	FB_AlarmCodeManager(	
		bAlarm1			:= MesDataExd.MesData.ProtectRelay_FeederMVCB[1].OUT_CmdOpen , 	// ProtectRelay_FeederMVCB Midi : Cmd Open
		bAlarm2			:= MesDataExd.MesData.ProtectRelay_FeederMVCB[1].OUT_CmdClose,     // ProtectRelay_FeederMVCB Midi  : Cmd Close
		bAlarm3			:= MesDataExd.MesData.ProtectRelay_FeederMVCB[2].OUT_CmdOpen  ,    // ProtectRelay_FeederMVCB Plat  : Cmd Open
		bAlarm4			:= MesDataExd.MesData.ProtectRelay_FeederMVCB[2].OUT_CmdClose ,	// ProtectRelay_FeederMVCB Plat  : Cmd Close
		bAlarm5			:= MesDataExd.MesData.TapChanger.OUT_CmdRampUp,					// 225 kV Regleur : Cmd Ramp Up
		bAlarm6			:= MesDataExd.MesData.TapChanger.OUT_CmdRampDown ,                 // 225 kV Regleur :	Cmd Ramp Down
		bAlarm7			:= MesDataExd.MesData.MesAuxHtOpenSectLine225kV	 ,				// Aux Ht : Sect Line 225 kV Open
		bAlarm8			:= MesDataExd.MesData.MesAuxHtCloseSectLine225kV	,               // Aux Ht : Sect Line 225 kV Close
		bAlarm9			:= MesDataExd.MesData.MesAuxHtTeleCondamnSl225kV	 ,				// Aux Ht : Tele Condamn Sl 225 kV 
		bAlarm10		:= MesDataExd.MesData.MesAuxHtDeTeleCondamnSl225kV,       		// Aux Ht : DeTele Condamn Sl 225 kV
		bAlarm11		:= MesDataExd.MesData.MesAuxHtTelecommandeRelestActif ,			// Aux Ht : Telecommande Relest Actif
		bAlarm12		:= MesDataExd.MesData.MesAuxHtTelecommandeRelestPassif,           // Aux Ht : Telecommande Relest Passif
		bAlarm13		:= FALSE,
		bAlarm14		:= FALSE,
		bAlarm15		:= FALSE,
		wAlarmCode		=>MesDataExd.MesData.MesEventCode2);	
		
		
	FB_AlarmCodeManager(
		bAlarm1			:= MesDataExd.MesData.MesAuxHtOpenSectMalt,				// Aux Ht Sect Malt : Open
		bAlarm2			:= MesDataExd.MesData.MesAuxHtCloseSectMalt,				// Aux Ht Sect Malt : Close
		bAlarm3			:= MesDataExd.MesData.MesAuxBtSyntOpenDistrib48VccJdb,		// Aux Bt Synt : Open Distrib 48 Vcc Jdb
		bAlarm4			:= MesDataExd.MesData.MesAuxBtSyntOpenDistrib48VccLocker,	// Aux Bt Synt : Open Distrib 48 Vcc Locker
		bAlarm5			:= MesDataExd.MesData.MesAuxBt400VPermutAutoStopMode	,	// Aux Bt 400 V Permut Auto Stop Mode				
		bAlarm6			:= MesDataExd.MesData.MesAuxBt400VPermutAutoNormalMode	 ,	// Aux Bt 400 V Permut Auto Normal Mode
		bAlarm7			:= MesDataExd.MesData.MesAuxBt400VPermutAutoSecoursMode,	// Aux Bt 400 V Permut Auto Secours Mode
		bAlarm8			:= MesDataExd.MesData.MesAuxBt400VPermutModeAuto	,		// Aux Bt 400 V Permut Mode Auto
		bAlarm9			:= MesDataExd.MesData.UPS_CE.MesOpened_CBRectifier	,		// UPC CE : Opened CB Rectifier
		bAlarm10		:= MesDataExd.MesData.UPS_CE.MesOpened_CBBatt		    ,	// UPC CE : Opened CB Batt
		bAlarm11		:= MesDataExd.MesData.UPS_CE.MesOpened_CBAntenna		 ,	// UPC CE : Opened CB Antenna
		bAlarm12		:= MesDataExd.MesData.UPS_TCM.MesOpened_CBRectifier	,	// UPC TCM : Opened CB Rectifier
		bAlarm13		:= MesDataExd.MesData.UPS_TCM.MesOpened_CBBatt	   	 ,		// UPC TCM : Opened CB Batt
		bAlarm14		:= MesDataExd.MesData.UPS_TCM.MesOpened_CBAntenna	  ,		// UPC TCM : Opened CB Antenna 
		bAlarm15		:= FALSE,//  
		wAlarmCode		=>MesDataExd.MesData.MesEventCode3);
END_METHOD

METHOD M_CP
//////////////////
//  Emulator
/////////////////

VAR 
	// Method local variables (reinitialized at each cycle) 
	

END_VAR
Trig_Cmd_Read(CLK:=IN_CmdToggleRead);


IF Trig_Cmd_Read.Q THEN
	IN_CmdToggleRead := FALSE;
MesDataExd.MesData.MesCP_Read := NOT MesDataExd.MesData.MesCP_Read;
END_IF
END_METHOD

METHOD M_Execute
//////////////////
//  Method Calls 
/////////////////
VAR 
	// Method local variables (reinitialized at each cycle) 
	// EMULATOR

	
END_VAR
// READING AND WRITING CLOCK //
	TP1(IN:=NOT TP1.Q , PT:= ParamClockReadTime);
	ClockRead 		:= TP1.Q;
	
// METHODS CALLS //

	M_Read() ; 
	M_CP();
	
// EVALUATE  /////////////
	

	
	////////////////////
	M_AlarmManagement();
END_METHOD

METHOD M_Read : BOOL
VAR_INPUT
END_VAR
VAR
	MW					: FB_MergeWordsToDint;
END_VAR
// CP-Read / Write 

MesDataExd.MesData.MesCP_Read := MesCP_Read ; 
MesDataExd.MesData.MesCP_Write := MesCP_Write ;  

IF MesCP_Read  THEN	

	// Analogic Inputs Modbus Requests
	
	FB_ModbusReadAI[1](pDestAddr := ADR(AI_List_1),
					sIPAddr := ParamIPAdr,
					tTimeout := ParamTimeout,
					nTcpPort := 502,
					nQuantity := 123,
					nMBAddr := 593,
					cbLength := SIZEOF(AI_List_1),
					nUnitID := 1,
					ClockRead := ClockRead,
					Reset := IN_CmdReset_L);
					
	FB_ModbusReadAI[2](pDestAddr := ADR(AI_List_2),
					sIPAddr := ParamIPAdr,
					tTimeout := ParamTimeout,
					nTcpPort := 502,
					nQuantity := 97,
					nMBAddr := 721,
					cbLength := SIZEOF(AI_List_2),
					nUnitID := 1,
					ClockRead := ClockRead,
					Reset := IN_CmdReset_L);
					
	// Digital Inputs Modbus Requests 
	
	FB_ModbusReadDI[1](pDestAddr := ADR(DI_List_1),
					sIPAddr := ParamIPAdr,
					tTimeout := ParamTimeout,
					nTcpPort := 502,
					nQuantity := 1683,
					nMBAddr := 480,
					cbLength := SIZEOF(DI_List_1),
					nUnitID := 1,
					ClockRead := ClockRead,
					Reset := IN_CmdReset_L);
					
	FB_ModbusReadDI[2](pDestAddr := ADR(DI_List_2),
					sIPAddr := ParamIPAdr,
					tTimeout := ParamTimeout,
					nTcpPort := 502,
					nQuantity := 1249,
					nMBAddr := 5072,
					cbLength := SIZEOF(DI_List_2),
					nUnitID := 1,
					ClockRead := ClockRead,
					Reset := IN_CmdReset_L);
	
					
					
	//  MesDataExd.MesData.Filling Digital Data				
	
MesDataExd.MesData.ProtectRelay_MainHVCB.MesAlarm_Phase1			:= DI_List_1[1]   ;
MesDataExd.MesData.ProtectRelay_MainHVCB.MesAlarm_Phase2		    := DI_List_1[2]   ;
MesDataExd.MesData.ProtectRelay_MainHVCB.MesAlarm_Phase3			:= DI_List_1[3]   ;
MesDataExd.MesData.ProtectRelay_MainHVCB.MesAlarm_PhaseRpt			:= DI_List_1[33]  ;
MesDataExd.MesData.ProtectRelay_MainHVCB.MesAlarm_Ground			:= DI_List_1[35]  ;
MesDataExd.MesData.ProtectRelay_MainHVCB.MesAlarm_GroundRpt		:= DI_List_1[36]  ;
MesDataExd.MesData.ProtectRelay_MainHVCB.MesAlarm_MaxUInverse		:= DI_List_1[37]  ;
MesDataExd.MesData.ProtectRelay_MainHVCB.MesAlarm_MaxP				:= DI_List_1[38]  ;
MesDataExd.MesData.ProtectRelay_MainHVCB.MesAlarm_CB				:= DI_List_1[39]  ;	
MesDataExd.MesData.ProtectRelay_MainHVCB.MesAlarm_Watchdog			:= DI_List_1[148] ;
	
				
	MesDataExd.MesData.ProtectRelay_Transfo225kV.MesAlarm_DiscordSectLigneHTB		   := DI_List_1[164]    ;
	MesDataExd.MesData.ProtectRelay_Transfo225kV.MesAlarm_DiscordSectMaltHTB         := DI_List_1[165]    ;
	MesDataExd.MesData.ProtectRelay_Transfo225kV.MesAlarm_DiscordSectDisjHTB         := DI_List_1[166]    ;
	MesDataExd.MesData.ProtectRelay_Transfo225kV.MesAlarm_TeleCondamne               := DI_List_1[167]    ;
	MesDataExd.MesData.ProtectRelay_Transfo225kV.MesAlarm_DeTeleCondamne             := DI_List_1[168]    ;
	MesDataExd.MesData.ProtectRelay_Transfo225kV.MesAlarm_DiscordTeleCondamne	       := DI_List_1[169]    ;
	MesDataExd.MesData.ProtectRelay_Transfo225kV.MesDataExd.MesData.MesAlarmImax                := DI_List_1[171]    ;
	MesDataExd.MesData.ProtectRelay_Transfo225kV.MesAlarm_IoMaxCoteProd              := DI_List_1[172]    ;
	MesDataExd.MesData.ProtectRelay_Transfo225kV.MesDataExd.MesData.MesAlarmUmin                := DI_List_1[173]    ;
	MesDataExd.MesData.ProtectRelay_Transfo225kV.MesDataExd.MesData.MesAlarmUmin_Long           := DI_List_1[174]    ;
	MesDataExd.MesData.ProtectRelay_Transfo225kV.MesAlarmUMax                        := DI_List_1[175]    ;
	MesDataExd.MesData.ProtectRelay_Transfo225kV.MesAlarmUMax_Long                   := DI_List_1[176]    ;
	MesDataExd.MesData.ProtectRelay_Transfo225kV.MesAlarm_PhaseRpt           	 	   := DI_List_1[177]    ;
	MesDataExd.MesData.ProtectRelay_Transfo225kV.MesWarning_ImgTherm                 := DI_List_1[178]    ;
	MesDataExd.MesData.ProtectRelay_Transfo225kV.MesAlarm_ImgTherm                   := DI_List_1[179]    ;
	MesDataExd.MesData.ProtectRelay_Transfo225kV.MesAlarm_DifferTransfo              := DI_List_1[180]    ;
	MesDataExd.MesData.ProtectRelay_Transfo225kV.MesAlarm_FreqMax                    := DI_List_1[181]    ;
	MesDataExd.MesData.ProtectRelay_Transfo225kV.MesAlarm_FreqMin                    := DI_List_1[183]    ;
	
	
	MesDataExd.MesData.MainHVCB.MesDataExd.MesData.MesClosed            				:= DI_List_1[193]    ;
	MesDataExd.MesData.MainHVCB.MesAlarm_SF6              				:= DI_List_1[197]    ;
	MesDataExd.MesData.MainHVCB.MesAlarm_Disarmed             	 		:= DI_List_1[198]    ;
	MesDataExd.MesData.MainHVCB.MesComutLocal         			   		:= DI_List_1[199]    ;
	MesDataExd.MesData.MainHVCB.MesAlarm_ArmingMotor           			:= DI_List_1[200]    ;
	MesDataExd.MesData.MainHVCB.MesAlarm_230V           					:= DI_List_1[201]    ;
	MesDataExd.MesData.MainHVCB.MesAlarmPwr          			 			:= DI_List_1[202]    ;
	
	MesDataExd.MesData.Transfo_225kV.MesWarningGas               			:= DI_List_1[220]    ;
	MesDataExd.MesData.Transfo_225kV.MesDataExd.MesData.MesAlarmGas           	 	:= DI_List_1[221]    ;
	MesDataExd.MesData.Transfo_225kV.MesDataExd.MesData.MesWarningTemp               := DI_List_1[222]    ;
	MesDataExd.MesData.Transfo_225kV.MesDataExd.MesData.MesAlarmGas             		:= DI_List_1[223]    ;
	MesDataExd.MesData.Transfo_225kV.MesWarning_TempLevel1           		:= DI_List_1[224]    ;
	MesDataExd.MesData.Transfo_225kV.MesWarning_TempLevel2          		:= DI_List_1[225]    ;
	MesDataExd.MesData.Transfo_225kV.MesTrigger_Deletion            		:= DI_List_1[228]    ;
	MesDataExd.MesData.Transfo_225kV.MesAlarm_OilLevel              		:= DI_List_1[229]    ;
	MesDataExd.MesData.Transfo_225kV.MesTransfoRefrigLocal                := DI_List_1[230]    ;
	MesDataExd.MesData.Transfo_225kV.MesTrigger_NonReturnValve       		:= DI_List_1[231]    ;
	MesDataExd.MesData.Transfo_225kV.MesTrigger_ProtectRelay      		:= DI_List_1[232]    ;
	MesDataExd.MesData.Transfo_225kV.MesAlarm_TapChanger            		:= DI_List_1[233]    ;
	
	MesDataExd.MesData.Mes20kVCourNeutCuveDefaultMasseCuve1		:= DI_List_1[305]	;
	MesDataExd.MesData.Mes20kVCourNeutCuveMaxIexp2				:= DI_List_1[306]   ;
	MesDataExd.MesData.Mes20kVCourNeutCuveDefaultMasseCuve2  		:= DI_List_1[307]   ;
	MesDataExd.MesData.Mes20kVCourNeutCuveMaxIexp4				:= DI_List_1[308]   ;
	MesDataExd.MesData.Mes20kVCourNeutCuveDefaultGround	    	:= DI_List_1[309]   ;
	MesDataExd.MesData.Mes20kVCourNeutCuveMaxI0exp4		    	:= DI_List_1[310]   ;
	MesDataExd.MesData.Mes20kVCourNeutCuveTempAlarm		    	:= DI_List_1[439]   ;
	MesDataExd.MesData.Mes20kVCourNeutCuveTempTrigger				:= DI_List_1[440]   ;
	MesDataExd.MesData.Mes20kVCourNeutCuveGazDischarge			:= DI_List_1[441]   ;
	MesDataExd.MesData.Mes20kVCourNeutCuvePressure           		:= DI_List_1[442]   ;
	
	MesDataExd.MesData.ProtectRelay_MainMVCB.MesAlarm_Phase1 			:= DI_List_1[457]	;
	MesDataExd.MesData.ProtectRelay_MainMVCB.MesAlarm_Phase2			:= DI_List_1[459]   ; // Phase 3  ? 
	MesDataExd.MesData.ProtectRelay_MainMVCB.MesAlarm_CB 				:= DI_List_1[495]   ;
	MesDataExd.MesData.ProtectRelay_MainMVCB.MesDataExd.MesData.MesTripped 		:= DI_List_1[586]   ; // Mes20kVGeneralHVCellProtectCircuitBreaker
	 /  MesDataExd.MesData.Mes20kVGeneralHVCellDefaultFrom225kV			:= DI_List_1[592]   ;
	
	MesDataExd.MesData.ProtectRelay_FeederMVCB[1].MesDataExd.MesData.MesAlarmImax 							:=	DI_List_1[609]	;
	MesDataExd.MesData.ProtectRelay_FeederMVCB[1].MesAlarm_MaxP									:=	DI_List_1[611]  ;
	MesDataExd.MesData.ProtectRelay_FeederMVCB[1].MesAlarm_Ground									:=	DI_List_1[613]  ;
	//  MesDataExd.MesData.AX_ProtectRelay_FeederMVCB[1].Mes20kVMidiSepamDefaultCablesOvercharge	:=	DI_List_1[641]  ;
	//  MesDataExd.MesData.AX_ProtectRelay_FeederMVCB[1].Mes20kVMidiHVCellDefaultFrom225kV			:=	DI_List_1[647]  ;
	MesDataExd.MesData.ProtectRelay_FeederMVCB[1].MesDataExd.MesData.MesTripped								:=	DI_List_1[738]  ;
	                                                                                	
	MesDataExd.MesData.ProtectRelay_FeederMVCB[2].MesDataExd.MesData.MesAlarmImax							:=	 DI_List_1[761] ;
	MesDataExd.MesData.ProtectRelay_FeederMVCB[2].MesAlarm_MaxP									:=   DI_List_1[763] ;
	MesDataExd.MesData.ProtectRelay_FeederMVCB[2].MesAlarm_Ground									:=   DI_List_1[765] ;  
	//  MesDataExd.MesData.AX_ProtectRelay_FeederMVCB[2].Mes20kVMidiSepamDefaultCablesOvercharge	:=   DI_List_1[793] ;
	//  MesDataExd.MesData.AX_ProtectRelay_FeederMVCB[2].Mes20kVMidiHVCellDefaultFrom225kV			:=   DI_List_1[799] ;
	MesDataExd.MesData.ProtectRelay_FeederMVCB[2].MesDataExd.MesData.MesTripped								:=   DI_List_1[890] ;
	
	MesDataExd.MesData.TapChanger.MesAlarm  := DI_List_1[1065] ;
	
	MesDataExd.MesData.MesAuxHTSect225kV							:=	DI_List_1[1217]	 ;
	MesDataExd.MesData.MesAuxHtSmaltHTBOpen						:=	DI_List_1[1219]	 ;
	MesDataExd.MesData.MesAuxHtFusionFuseMeasures225kV			:=	DI_List_1[1225]	 ;
	MesDataExd.MesData.MesAuxHtFusionFuseProtect225kV				:=	DI_List_1[1226]	 ;
	MesDataExd.MesData.MesAuxHtFusionFuseCountRte225kV			:=	DI_List_1[1227]	 ;
	MesDataExd.MesData.MesAuxHtShortCircuitCurrentProtectCcp2		:=	DI_List_1[1228]	 ;
	MesDataExd.MesData.MesAuxHtDisjCount20kVOpen					:=	DI_List_1[1230]	 ;
	MesDataExd.MesData.MesAuxHtDisjRefVoltage20kVOpen				:=	DI_List_1[1231]	 ;
	MesDataExd.MesData.MesAuxHtShortCircuitCurrentProtectCcp3		:=	DI_List_1[1232]	 ;
	MesDataExd.MesData.MesAuxBtTriggerGeneralDisj					:=	DI_List_1[1372]	 ;
	MesDataExd.MesData.MesAuxBt400VManqueAC						:=	DI_List_1[1373]	 ;
	MesDataExd.MesData.MesAuxBt400VDecltAntenneScada				:=	DI_List_1[1374]  ;
	MesDataExd.MesData.MesAuxBt400VDecltAntennePrio				:=	DI_List_1[1375]	 ;
	MesDataExd.MesData.MesAuxBt400VPermutAutoStopMode				:=	DI_List_1[1377]	 ;
	MesDataExd.MesData.MesAuxBt400VPermutAutoNormalMode			:=	DI_List_1[1378]	 ;
	MesDataExd.MesData.MesAuxBt400VPermutAutoSecoursMode			:=	DI_List_1[1379]	 ;
	MesDataExd.MesData.MesAuxBt400VPermutModeAuto					:=	DI_List_1[1380]	 ;
	MesDataExd.MesData.MesAuxBt400VVoltageLossNormalAlim			:=	DI_List_1[1381]	 ;
	MesDataExd.MesData.MesAuxBt400VVoltageLossSecoursAlim			:=	DI_List_1[1382]	 ;
	MesDataExd.MesData.MesAuxBt400VDefaultPermut					:=	DI_List_1[1383]	 ;
	
	
	
	MesDataExd.MesData.UPS_CE.MesAlarm_Batt 						:=	DI_List_1[1384]	 ;
	MesDataExd.MesData.UPS_CE.MesDataExd.MesData.MesAlarmState 				:=	DI_List_1[1385]	 ;
	MesDataExd.MesData.UPS_CE.MesAlarm_IsolBatt					:=	DI_List_1[1386]	 ;
	MesDataExd.MesData.UPS_CE.MesOpened_CBRectifier				:=	DI_List_1[1387]	 ;
	MesDataExd.MesData.UPS_CE.MesOpened_CBBatt					:=	DI_List_1[1388]	 ;
	MesDataExd.MesData.UPS_CE.MesOpened_CBAntenna					:=	DI_List_1[1389]	 ;
	MesDataExd.MesData.UPS_TCM.MesAlarm_Batt						:=	DI_List_1[1390]	 ;
	MesDataExd.MesData.UPS_TCM.MesDataExd.MesData.MesAlarmState				:=	DI_List_1[1391]	 ;
	MesDataExd.MesData.UPS_TCM.MesOpened_CBRectifier				:=	DI_List_1[1392]	 ;
	MesDataExd.MesData.UPS_TCM.MesOpened_CBBatt	   				:=	DI_List_1[1393]	 ;
	MesDataExd.MesData.UPS_TCM.MesOpened_CBAntenna				:=	DI_List_1[1394]	 ;
	 
	MesDataExd.MesData.MesAuxBtDefaultInverter					:=	DI_List_1[1395]	 ;
	MesDataExd.MesData.MesAuxBtSyntDefaultDistrib48VccJdb			:=	DI_List_1[1397]	 ;
	MesDataExd.MesData.MesAuxBtSyntOpenDistrib48VccJdb			:=	DI_List_1[1398]	 ;
	MesDataExd.MesData.MesAuxBtSyntDefaultDistrib48VccLocker		:=	DI_List_1[1403]	 ;
	MesDataExd.MesData.MesAuxBtSyntOpenDistrib48VccLocker			:=	DI_List_1[1404]	 ;
	 
	MesDataExd.MesData.Transfo_Aux.MesDataExd.MesData.MesAlarmTemp			:=	DI_List_1[1522]	 ;
	MesDataExd.MesData.Transfo_Aux.MesDataExd.MesData.MesAlarmGas			:=	DI_List_1[1523]	 ;
	MesDataExd.MesData.Transfo_Aux.MesDataExd.MesData.MesAlarmOilLevel		:=	DI_List_1[1524]	 ;
	 
	MesDataExd.MesData.MesAuxTransfoMeltingFusesContact			:=	DI_List_1[1525]	 ;                             
	MesDataExd.MesData.MesAuxTransfoSwitchGear	            	:=	DI_List_1[1526]  ;
	
	MesDataExd.MesData.DS.MesAlarmState          	  	:=	DI_List_1[1673] ;
	MesDataExd.MesData.FSS.MesAlarmFire				:=	DI_List_1[1674]	;
	MesDataExd.MesData.MesLocalRemoteOperation  	:=	DI_List_1[1682]	;
	MesDataExd.MesData.ES.MesAlarmState         		:=	DI_List_1[1683]	;
	 
	
						
	 /  MesDataExd.MesData.ProtectRelay_MainHVCB.MesDataExd.MesData.MesWatchdog 	  := DI_List_2[1]	; 
	MesDataExd.MesData.ProtectRelay_MainHVCB.MesDataExd.MesData.MesAlarmTCS    := DI_List_2[12]	;
	
	MesDataExd.MesData.ProtectRelay_Transfo225kV.MesDataExd.MesData.MesAlarmTCS 	 := DI_List_2[39] ;
	 // Mes225kVTransfoDefaultInternDisjCde := DI_List_2[46] ;
	
	MesDataExd.MesData.ProtectRelay_MainMVCB.MesDataExd.MesData.MesWatchdog 	 :=   DI_List_2[97]	; 
	MesDataExd.MesData.ProtectRelay_MainMVCB.MesDataExd.MesData.MesAlarmTCS   := 	DI_List_2[108]	;
	
	MesDataExd.MesData.ProtectRelay_FeederMVCB[1].MesDataExd.MesData.MesWatchdog   :=   DI_List_2[129] ;
	MesDataExd.MesData.ProtectRelay_FeederMVCB[1].MesDataExd.MesData.MesAlarmTCS   := 	 DI_List_2[140] ;
	
	MesDataExd.MesData.ProtectRelay_FeederMVCB[2].MesDataExd.MesData.MesWatchdog	  :=   DI_List_2[161]  ; 
	MesDataExd.MesData.ProtectRelay_FeederMVCB[2].MesDataExd.MesData.MesAlarmTCS   := 	 DI_List_2[172]  ;
	
	MesDataExd.MesData.TapChanger.MesAlarm_Discordance				  :=  DI_List_2[225]	;
	MesDataExd.MesData.TapChanger.MesAlarm_NoOutletDetected			  :=  DI_List_2[226]	;          
	MesDataExd.MesData.TapChanger.MesModeAuto							  :=  DI_List_2[227]	;
	MesDataExd.MesData.TapChanger.MesModeManual						  :=  DI_List_2[228]	;
	MesDataExd.MesData.TapChanger.MesState_ManoeuverAuthorized 		  :=  DI_List_2[230]	;
	
	MesDataExd.MesData.ProtectRelay_MainHVCB.OUT_CmdOpen  			  :=  DI_List_2[990] ;
	MesDataExd.MesData.ProtectRelay_MainHVCB.OUT_CmdClose     		  :=  DI_List_2[991] ;
	
	//  MesDataExd.MesData.Mes225kVTransfoDeclenchOpen	 := DI_List_2[1019] ;
	//  MesDataExd.MesData.Mes225kVTransfoEnclenchClose    := DI_List_2[1020] ;
	
	MesDataExd.MesData.ProtectRelay_MainMVCB.OUT_CmdOpen 	 :=  DI_List_2[1077] ;
	MesDataExd.MesData.ProtectRelay_MainMVCB.OUT_CmdClose  :=  DI_List_2[1078] ;
	
	MesDataExd.MesData.ProtectRelay_FeederMVCB[1].OUT_CmdOpen 	:=	DI_List_2[1106]  ; // MIDI 
	MesDataExd.MesData.ProtectRelay_FeederMVCB[1].OUT_CmdClose :=  DI_List_2[1107]  ;
	
	MesDataExd.MesData.ProtectRelay_FeederMVCB[2].OUT_CmdOpen   :=  DI_List_2[1135]	;	// PLAT 
	MesDataExd.MesData.ProtectRelay_FeederMVCB[2].OUT_CmdClose  :=  DI_List_2[1136]  ;
	
	MesDataExd.MesData.TapChanger.OUT_CmdRampUp	:=  DI_List_2[1193] ;
	MesDataExd.MesData.TapChanger.OUT_CmdRampDown :=	DI_List_2[1194] ;           
	MesDataExd.MesData.TapChanger.MesModeManual	:=  DI_List_2[1195]	;
	MesDataExd.MesData.TapChanger.MesModeAuto    :=  DI_List_2[1196] ;
	
	MesDataExd.MesData.MesAuxHtOpenSectLine225kV		  :=  DI_List_1[1242]  	;
	MesDataExd.MesData.MesAuxHtCloseSectLine225kV		  :=  DI_List_1[1243] 	;
	MesDataExd.MesData.MesAuxHtOpenSectMalt			  :=  DI_List_1[1244]   ;  
	MesDataExd.MesData.MesAuxHtCloseSectMalt			  :=  DI_List_1[1245]   ; 	
	MesDataExd.MesData.MesAuxHtTeleCondamnSl225kV		  :=  DI_List_1[1246] 	;
	MesDataExd.MesData.MesAuxHtDeTeleCondamnSl225kV	  :=  DI_List_1[1247]   ;                          
	MesDataExd.MesData.MesAuxHtTelecommandeRelestActif  :=  DI_List_1[1248]   ;
	MesDataExd.MesData.MesAuxHtTelecommandeRelestPassif :=  DI_List_1[1249]   ;
	
	//  MesDataExd.MesData.Filling Analogic Data			           
					                                
	MW(WORD_STRONG :=  AI_List_1[1  ],	WORD_WEAK := AI_List_1[1  ], SIZE := 1, FIX := 0, SIGNED := 0, VAR_OUT	:= MesDataExd.MesData.ProtectRelay_MainHVCB.MesDataExd.MesData.MesI1);
	MW(WORD_STRONG :=  AI_List_1[2  ],	WORD_WEAK := AI_List_1[2  ], SIZE := 1, FIX := 0, SIGNED := 0, VAR_OUT	:= MesDataExd.MesData.ProtectRelay_MainHVCB.MesDataExd.MesData.MesI2);
	MW(WORD_STRONG :=  AI_List_1[3  ],	WORD_WEAK := AI_List_1[3  ], SIZE := 1, FIX := 0, SIGNED := 0, VAR_OUT	:= MesDataExd.MesData.ProtectRelay_MainHVCB.MesDataExd.MesData.MesI3);
	MW(WORD_STRONG :=  AI_List_1[12 ],	WORD_WEAK := AI_List_1[12 ], SIZE := 1, FIX := 3, SIGNED := 0, VAR_OUT	:= MesDataExd.MesData.ProtectRelay_MainHVCB.MesDataExd.MesData.MesU12);
	MW(WORD_STRONG :=  AI_List_1[13 ],	WORD_WEAK := AI_List_1[13 ], SIZE := 1, FIX := 3, SIGNED := 0, VAR_OUT	:= MesDataExd.MesData.ProtectRelay_MainHVCB.MesDataExd.MesData.MesU23);
	MW(WORD_STRONG :=  AI_List_1[14 ],	WORD_WEAK := AI_List_1[14 ], SIZE := 1, FIX := 3, SIGNED := 0, VAR_OUT	:= MesDataExd.MesData.ProtectRelay_MainHVCB.MesDataExd.MesData.MesU31);
	MW(WORD_STRONG :=  AI_List_1[18 ],	WORD_WEAK := AI_List_1[18 ], SIZE := 1, FIX := 0, SIGNED := 0, VAR_OUT	:= MesDataExd.MesData.ProtectRelay_MainHVCB.MesU0);
	MW(WORD_STRONG :=  AI_List_1[21 ],	WORD_WEAK := AI_List_1[21 ], SIZE := 1, FIX := 0, SIGNED := 0, VAR_OUT	:= MesDataExd.MesData.ProtectRelay_MainHVCB.MesDataExd.MesData.MesFreq);
	MW(WORD_STRONG :=  AI_List_1[22 ],	WORD_WEAK := AI_List_1[22 ], SIZE := 1, FIX := 0, SIGNED := 0, VAR_OUT	:= MesDataExd.MesData.ProtectRelay_MainHVCB.MesP);
	MW(WORD_STRONG :=  AI_List_1[23 ],	WORD_WEAK := AI_List_1[23 ], SIZE := 1, FIX := 0, SIGNED := 0, VAR_OUT	:= MesDataExd.MesData.ProtectRelay_MainHVCB.MesQ);
	MW(WORD_STRONG :=  AI_List_1[27 ],	WORD_WEAK := AI_List_1[27 ], SIZE := 1, FIX := 0, SIGNED := 0, VAR_OUT	:= MesDataExd.MesData.ProtectRelay_MainHVCB.MesCosPhi);
	                               
	MW(WORD_STRONG :=  AI_List_1[33 ],	WORD_WEAK := AI_List_1[33 ], SIZE := 1, FIX := 0, SIGNED := 0, VAR_OUT	:= MesDataExd.MesData.ProtectRelay_Transfo225kV.MesDataExd.MesData.MesI1);
	MW(WORD_STRONG :=  AI_List_1[34 ],	WORD_WEAK := AI_List_1[34 ], SIZE := 1, FIX := 0, SIGNED := 0, VAR_OUT	:= MesDataExd.MesData.ProtectRelay_Transfo225kV.MesDataExd.MesData.MesI2);
	MW(WORD_STRONG :=  AI_List_1[35 ],	WORD_WEAK := AI_List_1[35 ], SIZE := 1, FIX := 0, SIGNED := 0, VAR_OUT	:= MesDataExd.MesData.ProtectRelay_Transfo225kV.MesDataExd.MesData.MesI3);
	MW(WORD_STRONG :=  AI_List_1[44 ],	WORD_WEAK := AI_List_1[44 ], SIZE := 1, FIX := 3, SIGNED := 0, VAR_OUT	:= MesDataExd.MesData.ProtectRelay_Transfo225kV.MesDataExd.MesData.MesU12);
	MW(WORD_STRONG :=  AI_List_1[45 ],	WORD_WEAK := AI_List_1[45 ], SIZE := 1, FIX := 3, SIGNED := 0, VAR_OUT	:= MesDataExd.MesData.ProtectRelay_Transfo225kV.MesDataExd.MesData.MesU23);
	MW(WORD_STRONG :=  AI_List_1[46 ],	WORD_WEAK := AI_List_1[46 ], SIZE := 1, FIX := 3, SIGNED := 0, VAR_OUT	:= MesDataExd.MesData.ProtectRelay_Transfo225kV.MesDataExd.MesData.MesU31);
	MW(WORD_STRONG :=  AI_List_1[54 ],	WORD_WEAK := AI_List_1[54 ], SIZE := 1, FIX := 0, SIGNED := 0, VAR_OUT	:= MesDataExd.MesData.ProtectRelay_Transfo225kV.MesP);
	MW(WORD_STRONG :=  AI_List_1[55 ],	WORD_WEAK := AI_List_1[55 ], SIZE := 1, FIX := 0, SIGNED := 0, VAR_OUT	:= MesDataExd.MesData.ProtectRelay_Transfo225kV.MesQ);
	
	MW(WORD_STRONG :=  AI_List_1[65 ],	WORD_WEAK := AI_List_1[65 ], SIZE := 1, FIX := 0, SIGNED := 0, VAR_OUT	:= MesDataExd.MesData.Mes20kVCourNeutCuveI1);
	MW(WORD_STRONG :=  AI_List_1[69 ],	WORD_WEAK := AI_List_1[69 ], SIZE := 1, FIX := 0, SIGNED := 0, VAR_OUT	:= MesDataExd.MesData.Mes20kVCourNeutCuveResidualI);
	MW(WORD_STRONG :=  AI_List_1[92 ],	WORD_WEAK := AI_List_1[92 ], SIZE := 1, FIX := 0, SIGNED := 0, VAR_OUT	:= MesDataExd.MesData.Mes20kVCourNeutCuveDecltI1);
	MW(WORD_STRONG :=  AI_List_1[95 ],	WORD_WEAK := AI_List_1[95 ], SIZE := 1, FIX := 0, SIGNED := 0, VAR_OUT	:= MesDataExd.MesData.Mes20kVCourNeutCuveDecltI2);
	
	MW(WORD_STRONG :=  AI_List_1[97  ],	WORD_WEAK := AI_List_1[97  ], SIZE := 1, FIX := 0, SIGNED := 0, VAR_OUT	:= MesDataExd.MesData.ProtectRelay_MainMVCB.MesDataExd.MesData.MesI1);
	MW(WORD_STRONG :=  AI_List_1[98  ],	WORD_WEAK := AI_List_1[98  ], SIZE := 1, FIX := 0, SIGNED := 0, VAR_OUT	:= MesDataExd.MesData.ProtectRelay_MainMVCB.MesDataExd.MesData.MesI2);
	MW(WORD_STRONG :=  AI_List_1[99  ],	WORD_WEAK := AI_List_1[99  ], SIZE := 1, FIX := 0, SIGNED := 0, VAR_OUT	:= MesDataExd.MesData.ProtectRelay_MainMVCB.MesDataExd.MesData.MesI3);
	MW(WORD_STRONG :=  AI_List_1[108 ],	WORD_WEAK := AI_List_1[108 ], SIZE := 1, FIX := 3, SIGNED := 0, VAR_OUT	:= MesDataExd.MesData.ProtectRelay_MainMVCB.MesDataExd.MesData.MesU12);
	MW(WORD_STRONG :=  AI_List_1[109 ],	WORD_WEAK := AI_List_1[109 ], SIZE := 1, FIX := 3, SIGNED := 0, VAR_OUT	:= MesDataExd.MesData.ProtectRelay_MainMVCB.MesDataExd.MesData.MesU23);
	MW(WORD_STRONG :=  AI_List_1[110 ],	WORD_WEAK := AI_List_1[110 ], SIZE := 1, FIX := 3, SIGNED := 0, VAR_OUT	:= MesDataExd.MesData.ProtectRelay_MainMVCB.MesDataExd.MesData.MesU31);
	MW(WORD_STRONG :=  AI_List_1[114 ],	WORD_WEAK := AI_List_1[114 ], SIZE := 1, FIX := 0, SIGNED := 0, VAR_OUT	:= MesDataExd.MesData.ProtectRelay_MainMVCB.MesU0);
	MW(WORD_STRONG :=  AI_List_1[117 ],	WORD_WEAK := AI_List_1[117 ], SIZE := 1, FIX := 0, SIGNED := 0, VAR_OUT	:= MesDataExd.MesData.ProtectRelay_MainMVCB.MesDataExd.MesData.MesFreq);
	MW(WORD_STRONG :=  AI_List_1[119 ],	WORD_WEAK := AI_List_1[119 ], SIZE := 1, FIX := 0, SIGNED := 0, VAR_OUT	:= MesDataExd.MesData.ProtectRelay_MainMVCB.MesP);
	MW(WORD_STRONG :=  AI_List_1[120 ],	WORD_WEAK := AI_List_1[120 ], SIZE := 1, FIX := 0, SIGNED := 0, VAR_OUT	:= MesDataExd.MesData.ProtectRelay_MainMVCB.MesQ);
	MW(WORD_STRONG :=  AI_List_1[123 ],	WORD_WEAK := AI_List_1[123 ], SIZE := 1, FIX := 0, SIGNED := 0, VAR_OUT	:= MesDataExd.MesData.ProtectRelay_MainMVCB.MesCosPhi);
	
	MW(WORD_STRONG :=  AI_List_2[1 	 ], WORD_WEAK := AI_List_2[1 ], SIZE := 1, FIX := 0, SIGNED := 0, VAR_OUT	:= MesDataExd.MesData.ProtectRelay_FeederMVCB[1].MesDataExd.MesData.MesI1);
	MW(WORD_STRONG :=  AI_List_2[2   ], WORD_WEAK := AI_List_2[2 ], SIZE := 1, FIX := 0, SIGNED := 0, VAR_OUT	:= MesDataExd.MesData.ProtectRelay_FeederMVCB[1].MesDataExd.MesData.MesI2);
	MW(WORD_STRONG :=  AI_List_2[3   ], WORD_WEAK := AI_List_2[3 ], SIZE := 1, FIX := 0, SIGNED := 0, VAR_OUT	:= MesDataExd.MesData.ProtectRelay_FeederMVCB[1].MesDataExd.MesData.MesI3);
	MW(WORD_STRONG :=  AI_List_2[22  ], WORD_WEAK := AI_List_2[22 ], SIZE := 1, FIX := 0, SIGNED := 0, VAR_OUT	:= MesDataExd.MesData.ProtectRelay_FeederMVCB[1].MesP);
	MW(WORD_STRONG :=  AI_List_2[23  ], WORD_WEAK := AI_List_2[23 ], SIZE := 1, FIX := 0, SIGNED := 0, VAR_OUT	:= MesDataExd.MesData.ProtectRelay_FeederMVCB[1].MesQ);
	                                                        
	MW(WORD_STRONG :=  AI_List_2[33 ], WORD_WEAK := AI_List_2[33 ], SIZE := 1, FIX := 0, SIGNED := 0, VAR_OUT	:= MesDataExd.MesData.ProtectRelay_FeederMVCB[2].MesDataExd.MesData.MesI1);
	MW(WORD_STRONG :=  AI_List_2[34 ], WORD_WEAK := AI_List_2[34 ], SIZE := 1, FIX := 0, SIGNED := 0, VAR_OUT	:= MesDataExd.MesData.ProtectRelay_FeederMVCB[2].MesDataExd.MesData.MesI2);
	MW(WORD_STRONG :=  AI_List_2[35 ], WORD_WEAK := AI_List_2[35 ], SIZE := 1, FIX := 0, SIGNED := 0, VAR_OUT	:= MesDataExd.MesData.ProtectRelay_FeederMVCB[2].MesDataExd.MesData.MesI3);
	MW(WORD_STRONG :=  AI_List_2[54 ], WORD_WEAK := AI_List_2[54 ], SIZE := 1, FIX := 0, SIGNED := 0, VAR_OUT	:= MesDataExd.MesData.ProtectRelay_FeederMVCB[2].MesP);         
	MW(WORD_STRONG :=  AI_List_2[55 ], WORD_WEAK := AI_List_2[55 ], SIZE := 1, FIX := 0, SIGNED := 0, VAR_OUT	:= MesDataExd.MesData.ProtectRelay_FeederMVCB[2].MesQ);         

END_IF
//MW(WORD_STRONG :=  AI_List_2[97 ], WORD_WEAK := AI_List_2[97 ], SIZE := 1, FIX := 0, SIGNED := 0, VAR_OUT	:= MesDataExd.MesData.Mes20kVPlatSepamQ);	






(*			
//  MesDataExd.MesData.Filling Digital Data				

MesData.Mes225kVCombiDefaultPhase1			:= DI_List_1[1]   ;
MesData.Mes225kVCombiDefaultPhase2		    := DI_List_1[2]   ;
MesData.Mes225kVCombiDefaultPhase3			:= DI_List_1[3]   ;
MesData.Mes225kVCombiDefaultPhaseRpt		:= DI_List_1[33]  ;
MesData.Mes225kVCombiDefaultGround			:= DI_List_1[35]  ;
MesData.Mes225kVCombiDefaultGroundRpt		:= DI_List_1[36]  ;
MesData.Mes225kVCombiDefaultMaxUInverse		:= DI_List_1[37]  ;
MesData.Mes225kVCombiDefaultMaxP			:= DI_List_1[38]  ;
MesData.Mes225kVCombiDefaultCircuitbreaker	:= DI_List_1[39]  ;	
MesData.Mes225kVCombiDefaultWatchdog		:= DI_List_1[148] ;
			
MesDataExd.MesData.Mes225kVTransfoDiscordSectLigneHTB		   := DI_List_1[164]    ;
MesDataExd.MesData.Mes225kVTransfoDiscordSectMaltHTB         := DI_List_1[165]    ;
MesDataExd.MesData.Mes225kVTransfoDiscordSectDisjHTB         := DI_List_1[166]    ;
MesDataExd.MesData.Mes225kVTransfoTeleCondamne               := DI_List_1[167]    ;
MesDataExd.MesData.Mes225kVTransfoDeTeleCondamne             := DI_List_1[168]    ;
MesDataExd.MesData.Mes225kVTransfoDiscordTeleCondamne	       := DI_List_1[169]    ;
MesDataExd.MesData.Mes225kVTransfoMaxI	                   := DI_List_1[170]    ;
MesDataExd.MesData.Mes225kVTransfoMaxICoteProd               := DI_List_1[171]    ;
MesDataExd.MesData.Mes225kVTransfoMaxIoCoteProd              := DI_List_1[172]    ;
MesDataExd.MesData.Mes225kVTransfoMinU                       := DI_List_1[173]    ;
MesDataExd.MesData.Mes225kVTransfoMinULong                   := DI_List_1[174]    ;
MesDataExd.MesData.Mes225kVTransfoMaxU                       := DI_List_1[175]    ;
MesDataExd.MesData.Mes225kVTransfoMaxULong                   := DI_List_1[176]    ;
MesDataExd.MesData.Mes225kVTransfoDefaultPhaseRpt            := DI_List_1[177]    ;
MesDataExd.MesData.Mes225kVTransfoAlarmImgTherm              := DI_List_1[178]    ;
MesDataExd.MesData.Mes225kVTransfoDefaultImgTherm            := DI_List_1[179]    ;
MesDataExd.MesData.Mes225kVTransfoDifferTransfo              := DI_List_1[180]    ;
MesDataExd.MesData.Mes225kVTransfoMaxFreq                    := DI_List_1[181]    ;
MesDataExd.MesData.Mes225kVTransfoMinFreq                    := DI_List_1[183]    ;
MesDataExd.MesData.Mes225kVTransfoCircuitBreaker             := DI_List_1[193]    ;
MesDataExd.MesData.Mes225kVTransfoDisjManqueSf6              := DI_List_1[197]    ;
MesDataExd.MesData.Mes225kVTransfoCmdDisjDesarm              := DI_List_1[198]    ;
MesDataExd.MesData.Mes225kVTransfoCmdDisjDistVerr            := DI_List_1[199]    ;
MesDataExd.MesData.Mes225kVTransfoDefaultMoteurArm           := DI_List_1[200]    ;
MesDataExd.MesData.Mes225kVTransfoDefaultAux230Vac           := DI_List_1[201]    ;
MesDataExd.MesData.Mes225kVTransfoDefaultAlimBobine          := DI_List_1[202]    ;
MesDataExd.MesData.Mes225kVTransfoAlarmBuchholz              := DI_List_1[220]    ;
MesDataExd.MesData.Mes225kVTransfoTriggerBuchHolz            := DI_List_1[221]    ;
MesDataExd.MesData.Mes225kVTransfoAlarmTempOil               := DI_List_1[222]    ;
MesDataExd.MesData.Mes225kVTransfoTriggerTempOil             := DI_List_1[223]    ;
MesDataExd.MesData.Mes225kVTransfoImgTherm1erStade           := DI_List_1[224]    ;
MesDataExd.MesData.Mes225kVTransfoImgTherm2emeStade          := DI_List_1[225]    ;
MesDataExd.MesData.Mes225kVTransfoDcltSurpression            := DI_List_1[228]    ;
MesDataExd.MesData.Mes225kVTransfoNiveauMiniOil              := DI_List_1[229]    ;
MesDataExd.MesData.Mes225kVTransfoRefrigLocal                := DI_List_1[230]    ;
MesDataExd.MesData.Mes225kVTransfoDcltClapetAntiRetour       := DI_List_1[231]    ;
MesDataExd.MesData.Mes225kVTransfoDcltRelaisProtectRegl      := DI_List_1[232]    ;
MesDataExd.MesData.Mes225kVTransfoDefaillanceRegl            := DI_List_1[233]    ;

MesDataExd.MesData.Mes20kVCourNeutCuveDefaultMasseCuve1		:= DI_List_1[305]	;
MesDataExd.MesData.Mes20kVCourNeutCuveMaxIexp2				:= DI_List_1[306]   ;
MesDataExd.MesData.Mes20kVCourNeutCuveDefaultMasseCuve2  		:= DI_List_1[307]   ;
MesDataExd.MesData.Mes20kVCourNeutCuveMaxIexp4				:= DI_List_1[308]   ;
MesDataExd.MesData.Mes20kVCourNeutCuveDefaultGround	    	:= DI_List_1[309]   ;
MesDataExd.MesData.Mes20kVCourNeutCuveMaxI0exp4		    	:= DI_List_1[310]   ;
MesDataExd.MesData.Mes20kVCourNeutCuveTempAlarm		    	:= DI_List_1[439]   ;
MesDataExd.MesData.Mes20kVCourNeutCuveTempTrigger				:= DI_List_1[440]   ;
MesDataExd.MesData.Mes20kVCourNeutCuveGazDischarge			:= DI_List_1[441]   ;
MesDataExd.MesData.Mes20kVCourNeutCuvePressure           		:= DI_List_1[442]   ;

MesDataExd.MesData.Mes20kVGeneralSepamDefaultPhase1			:= DI_List_1[457]	;
MesDataExd.MesData.Mes20kVGeneralSepamDefaultPhase2			:= DI_List_1[459]   ;
MesDataExd.MesData.Mes20kVGeneralHVCellDefaultCircuitBreaker	:= DI_List_1[495]   ;
MesDataExd.MesData.Mes20kVGeneralHVCellProtectCircuitBreaker	:= DI_List_1[586]   ;
MesDataExd.MesData.Mes20kVGeneralHVCellDefaultFrom225kV		:= DI_List_1[592]   ;

MesDataExd.MesData.Mes20kVMidiSepamDefaultShortCircuit		:=	DI_List_1[609]	;
MesDataExd.MesData.Mes20kVMidiSepamDefaultOvercharge			:=	DI_List_1[611]  ;
MesDataExd.MesData.Mes20kVMidiSepamDefaultGround				:=	DI_List_1[613]  ;
MesDataExd.MesData.Mes20kVMidiSepamDefaultCablesOvercharge	:=	DI_List_1[641]  ;
MesDataExd.MesData.Mes20kVMidiHVCellDefaultFrom225kV			:=	DI_List_1[647]  ;
MesDataExd.MesData.Mes20kVMidiHVCellProtectCircuitBreaker		:=	DI_List_1[738]  ;

MesDataExd.MesData.Mes20kVPlatSepamDefaultShortCircuit		:=	 DI_List_1[761] ;
MesDataExd.MesData.Mes20kVPlatSepamDefaultOvercharge		 	:=   DI_List_1[763] ;
MesDataExd.MesData.Mes20kVPlatSepamDefaultGround			 	:=   DI_List_1[765] ;  
MesDataExd.MesData.Mes20kVPlatSepamDefaultCablesOvercharge	:=   DI_List_1[793] ;
MesDataExd.MesData.Mes20kVPlatHVCellDefaultFrom225kV		 	:=   DI_List_1[799] ;
MesDataExd.MesData.Mes20kVPlatHVCellProtectCircuitBreaker     :=   DI_List_1[890] ;

MesDataExd.MesData.Mes225kVRegleurDefault := DI_List_1[1065] ;

MesDataExd.MesData.MesAuxHTSect225kV							:=	DI_List_1[1217]	 ;
MesDataExd.MesData.MesAuxHtSmaltHTBOpen						:=	DI_List_1[1219]	 ;
MesDataExd.MesData.MesAuxHtFusionFuseMeasures225kV			:=	DI_List_1[1225]	 ;
MesDataExd.MesData.MesAuxHtFusionFuseProtect225kV				:=	DI_List_1[1226]	 ;
MesDataExd.MesData.MesAuxHtFusionFuseCountRte225kV			:=	DI_List_1[1227]	 ;
MesDataExd.MesData.MesAuxHtShortCircuitCurrentProtectCcp2		:=	DI_List_1[1228]	 ;
MesDataExd.MesData.MesAuxHtDisjCount20kVOpen					:=	DI_List_1[1230]	 ;
MesDataExd.MesData.MesAuxHtDisjRefVoltage20kVOpen				:=	DI_List_1[1231]	 ;
MesDataExd.MesData.MesAuxHtShortCircuitCurrentProtectCcp3		:=	DI_List_1[1232]	 ;
MesDataExd.MesData.MesAuxBtTriggerGeneralDisj					:=	DI_List_1[1372]	 ;
MesDataExd.MesData.MesAuxBt400VManqueAC						:=	DI_List_1[1373]	 ;
MesDataExd.MesData.MesAuxBt400VDecltAntenneScada				:=	DI_List_1[1374]  ;
MesDataExd.MesData.MesAuxBt400VDecltAntennePrio				:=	DI_List_1[1375]	 ;
MesDataExd.MesData.MesAuxBt400VPermutAutoStopMode				:=	DI_List_1[1377]	 ;
MesDataExd.MesData.MesAuxBt400VPermutAutoNormalMode			:=	DI_List_1[1378]	 ;
MesDataExd.MesData.MesAuxBt400VPermutAutoSecoursMode			:=	DI_List_1[1379]	 ;
MesDataExd.MesData.MesAuxBt400VPermutModeAuto					:=	DI_List_1[1380]	 ;
MesDataExd.MesData.MesAuxBt400VVoltageLossNormalAlim			:=	DI_List_1[1381]	 ;
MesDataExd.MesData.MesAuxBt400VVoltageLossSecoursAlim			:=	DI_List_1[1382]	 ;
MesDataExd.MesData.MesAuxBt400VDefaultPermut					:=	DI_List_1[1383]	 ;
MesDataExd.MesData.MesAuxBt48VCeDefaultBatt					:=	DI_List_1[1384]	 ;
MesDataExd.MesData.MesAuxBt48VCeDefaultRedress				:=	DI_List_1[1385]	 ;
MesDataExd.MesData.MesAuxBt48VCeDefaultIsolBatt				:=	DI_List_1[1386]	 ;
MesDataExd.MesData.MesAuxBt48VCeDecltDisjRedress				:=	DI_List_1[1387]	 ;
MesDataExd.MesData.MesAuxBt48VCeDecltDisjBatt					:=	DI_List_1[1388]	 ;
MesDataExd.MesData.MesAuxBt48VCeDecltAntenne					:=	DI_List_1[1389]	 ;
MesDataExd.MesData.MesAuxBt48VTcmDefaultBatt					:=	DI_List_1[1390]	 ;
MesDataExd.MesData.MesAuxBt48VTcmDefaultRedress				:=	DI_List_1[1391]	 ;
MesDataExd.MesData.MesAuxBt48VTcmDecltDisjRedress				:=	DI_List_1[1392]	 ;
MesDataExd.MesData.MesAuxBt48VTcmDecltDisjBatt				:=	DI_List_1[1393]	 ;
MesDataExd.MesData.MesAuxBt48VTcmDecltAntenne					:=	DI_List_1[1394]	 ;
MesDataExd.MesData.MesAuxBtDefaultInverter					:=	DI_List_1[1395]	 ;
MesDataExd.MesData.MesAuxBtSyntDefaultDistrib48VccJdb			:=	DI_List_1[1397]	 ;
MesDataExd.MesData.MesAuxBtSyntOpenDistrib48VccJdb			:=	DI_List_1[1398]	 ;
MesDataExd.MesData.MesAuxBtSyntDefaultDistrib48VccLocker		:=	DI_List_1[1403]	 ;
MesDataExd.MesData.MesAuxBtSyntOpenDistrib48VccLocker			:=	DI_List_1[1404]	 ;
MesDataExd.MesData.MesAuxTransfoTempTrigger					:=	DI_List_1[1522]	 ;
MesDataExd.MesData.MesAuxTransfoGazDischarge					:=	DI_List_1[1523]	 ;
MesDataExd.MesData.MesAuxTransfoPressure						:=	DI_List_1[1524]	 ;
MesDataExd.MesData.MesAuxTransfoMeltingFusesContact			:=	DI_List_1[1525]	 ;                             
MesDataExd.MesData.MesAuxTransfoSwitchGear	            	:=	DI_List_1[1526]  ;

MesDataExd.MesData.MesPDLDoorsOpen         	  	:=	DI_List_1[1673]	;
MesDataExd.MesData.MesPDLFireDetectorSystem    	:=	DI_List_1[1674]	;
MesDataExd.MesData.MesPDLLocalRemoteOperation  	:=	DI_List_1[1682]	;
MesDataExd.MesData.MesPDLEmergencyStop         	:=	DI_List_1[1683]	;
					
MesDataExd.MesData.Mes225kVCombiWatchdog		 := DI_List_2[1]	; 
MesDataExd.MesData.Mes225kVCombiDefaultMajor   := DI_List_2[12]	;

MesDataExd.MesData.Mes225kVTransfoSepamMajorDefault	 := DI_List_2[39] ;
MesDataExd.MesData.Mes225kVTransfoDefaultInternDisjCde := DI_List_2[46] ;

MesDataExd.MesData.Mes20kVGeneralSepamWatchdog	   :=   DI_List_2[97]	; 
MesDataExd.MesData.Mes20kVGeneralSepamDefaultMajor   := 	DI_List_2[108]	;

MesDataExd.MesData.Mes20kVMidiSepamWatchdog		:=   DI_List_2[129] ;
MesDataExd.MesData.Mes20kVMidiSepamDefaultMajor   := 	 DI_List_2[140] ;

MesDataExd.MesData.Mes20kVPlatSepamWatchdog		:=   DI_List_2[161]  ; 
MesDataExd.MesData.Mes20kVPlatSepamDefaultMajor   := 	 DI_List_2[172]  ;

MesDataExd.MesData.Mes225kVRegleurDefaultDiscordance	:=  DI_List_2[225]	;
MesDataExd.MesData.Mes225kVRegleurNoOutletDetected	:=	DI_List_2[226]	;          
MesDataExd.MesData.Mes225kVRegleurRegleurModeAuto		:=	DI_List_2[227]	;
MesDataExd.MesData.Mes225kVRegleurRegleurModeManuel	:=  DI_List_2[228]	;
MesDataExd.MesData.Mes225kVRegleurManoeuverAuthorized :=  DI_List_2[230]	;

MesDataExd.MesData.Mes225kVCombiOrderOpenCircuitBreaker 	:=  DI_List_2[990] ;
MesDataExd.MesData.Mes225kVCombiOrderCloseCircuitBreaker  :=  DI_List_2[991] ;

MesDataExd.MesData.Mes225kVTransfoDeclenchOpen	 := DI_List_2[1019] ;
MesDataExd.MesData.Mes225kVTransfoEnclenchClose    := DI_List_2[1020] ;

MesDataExd.MesData.Mes20kVGeneralHVCellProtectOrderOpenCircuitBreaker	 :=  DI_List_2[1077] ;
MesDataExd.MesData.Mes20kVGeneralHVCellProtectOrderCloseCircuitBreaker :=  DI_List_2[1078] ;

MesDataExd.MesData.Mes20kVMidiHVCellProtectOrderOpenCircuitBreaker	:=	DI_List_2[1106]  ;
MesDataExd.MesData.Mes20kVMidiHVCellProtectOrderCloseCircuitBreaker   :=  DI_List_2[1107]  ;

MesDataExd.MesData.Mes20kVPlatHVCellProtectOrderOpenCircuitBreaker   :=  DI_List_2[1135]	;
MesDataExd.MesData.Mes20kVPlatHVCellProtectOrderCloseCircuitBreaker  :=  DI_List_2[1136]  ;

MesDataExd.MesData.Mes225kVRegleurCdeMontee	:=  DI_List_2[1193] ;
MesDataExd.MesData.Mes225kVRegleurCdeDescente :=	DI_List_2[1194] ;           
MesDataExd.MesData.Mes225kVRegleurModeManuel	:=  DI_List_2[1195]	;
MesDataExd.MesData.Mes225kVRegleurModeAuto    :=  DI_List_2[1196] ;

MesDataExd.MesData.MesAuxHtOpenSectLine225kV		  :=  DI_List_1[1242]  	;
MesDataExd.MesData.MesAuxHtCloseSectLine225kV		  :=  DI_List_1[1243] 	;
MesDataExd.MesData.MesAuxHtOpenSectMalt			  :=  DI_List_1[1244]   ;  
MesDataExd.MesData.MesAuxHtCloseSectMalt			  :=  DI_List_1[1245]   ; 	
MesDataExd.MesData.MesAuxHtTeleCondamnSl225kV		  :=  DI_List_1[1246] 	;
MesDataExd.MesData.MesAuxHtDeTeleCondamnSl225kV	  :=  DI_List_1[1247]   ;                          
MesDataExd.MesData.MesAuxHtTelecommandeRelestActif  :=  DI_List_1[1248]   ;
MesDataExd.MesData.MesAuxHtTelecommandeRelestPassif :=  DI_List_1[1249]   ;

//  MesDataExd.MesData.Filling Analogic Data			           
				                                
MW(WORD_STRONG :=  AI_List_1[1  ],	WORD_WEAK := AI_List_1[1  ], SIZE := 1, FIX := 0, SIGNED := 0, VAR_OUT	:= MesDataExd.MesData.Mes225kVCombiI1);
MW(WORD_STRONG :=  AI_List_1[2  ],	WORD_WEAK := AI_List_1[2  ], SIZE := 1, FIX := 0, SIGNED := 0, VAR_OUT	:= MesDataExd.MesData.Mes225kVCombiI2);
MW(WORD_STRONG :=  AI_List_1[3  ],	WORD_WEAK := AI_List_1[3  ], SIZE := 1, FIX := 0, SIGNED := 0, VAR_OUT	:= MesDataExd.MesData.Mes225kVCombiI3);
MW(WORD_STRONG :=  AI_List_1[12 ],	WORD_WEAK := AI_List_1[12 ], SIZE := 1, FIX := 3, SIGNED := 0, VAR_OUT	:= MesDataExd.MesData.Mes225kVCombiU21);
MW(WORD_STRONG :=  AI_List_1[13 ],	WORD_WEAK := AI_List_1[13 ], SIZE := 1, FIX := 3, SIGNED := 0, VAR_OUT	:= MesDataExd.MesData.Mes225kVCombiU32);
MW(WORD_STRONG :=  AI_List_1[14 ],	WORD_WEAK := AI_List_1[14 ], SIZE := 1, FIX := 3, SIGNED := 0, VAR_OUT	:= MesDataExd.MesData.Mes225kVCombiU13);
MW(WORD_STRONG :=  AI_List_1[18 ],	WORD_WEAK := AI_List_1[18 ], SIZE := 1, FIX := 0, SIGNED := 0, VAR_OUT	:= MesDataExd.MesData.Mes225kVCombiResidualU);
MW(WORD_STRONG :=  AI_List_1[21 ],	WORD_WEAK := AI_List_1[21 ], SIZE := 1, FIX := 0, SIGNED := 0, VAR_OUT	:= MesDataExd.MesData.Mes225kVCombiFrequency);
MW(WORD_STRONG :=  AI_List_1[22 ],	WORD_WEAK := AI_List_1[22 ], SIZE := 1, FIX := 0, SIGNED := 0, VAR_OUT	:= MesDataExd.MesData.Mes225kVCombiP);
MW(WORD_STRONG :=  AI_List_1[23 ],	WORD_WEAK := AI_List_1[23 ], SIZE := 1, FIX := 0, SIGNED := 0, VAR_OUT	:= MesDataExd.MesData.Mes225kVCombiQ);
MW(WORD_STRONG :=  AI_List_1[27 ],	WORD_WEAK := AI_List_1[27 ], SIZE := 1, FIX := 0, SIGNED := 0, VAR_OUT	:= MesDataExd.MesData.Mes225kVCombiCosPhi);
                               
MW(WORD_STRONG :=  AI_List_1[33 ],	WORD_WEAK := AI_List_1[33 ], SIZE := 1, FIX := 0, SIGNED := 0, VAR_OUT	:= MesDataExd.MesData.Mes225kVTransfoI1);
MW(WORD_STRONG :=  AI_List_1[34 ],	WORD_WEAK := AI_List_1[34 ], SIZE := 1, FIX := 0, SIGNED := 0, VAR_OUT	:= MesDataExd.MesData.Mes225kVTransfoI2);
MW(WORD_STRONG :=  AI_List_1[35 ],	WORD_WEAK := AI_List_1[35 ], SIZE := 1, FIX := 0, SIGNED := 0, VAR_OUT	:= MesDataExd.MesData.Mes225kVTransfoI3);
MW(WORD_STRONG :=  AI_List_1[44 ],	WORD_WEAK := AI_List_1[44 ], SIZE := 1, FIX := 3, SIGNED := 0, VAR_OUT	:= MesDataExd.MesData.Mes225kVTransfoU21);
MW(WORD_STRONG :=  AI_List_1[45 ],	WORD_WEAK := AI_List_1[45 ], SIZE := 1, FIX := 3, SIGNED := 0, VAR_OUT	:= MesDataExd.MesData.Mes225kVTransfoU32);
MW(WORD_STRONG :=  AI_List_1[46 ],	WORD_WEAK := AI_List_1[46 ], SIZE := 1, FIX := 3, SIGNED := 0, VAR_OUT	:= MesDataExd.MesData.Mes225kVTransfoU13);
MW(WORD_STRONG :=  AI_List_1[54 ],	WORD_WEAK := AI_List_1[54 ], SIZE := 1, FIX := 0, SIGNED := 0, VAR_OUT	:= MesDataExd.MesData.Mes225kVTransfoP);
MW(WORD_STRONG :=  AI_List_1[55 ],	WORD_WEAK := AI_List_1[55 ], SIZE := 1, FIX := 0, SIGNED := 0, VAR_OUT	:= MesDataExd.MesData.Mes225kVTransfoQ);

MW(WORD_STRONG :=  AI_List_1[65 ],	WORD_WEAK := AI_List_1[65 ], SIZE := 1, FIX := 0, SIGNED := 0, VAR_OUT	:= MesDataExd.MesData.Mes20kVCourNeutCuveI1);
MW(WORD_STRONG :=  AI_List_1[69 ],	WORD_WEAK := AI_List_1[69 ], SIZE := 1, FIX := 0, SIGNED := 0, VAR_OUT	:= MesDataExd.MesData.Mes20kVCourNeutCuveResidualI);
MW(WORD_STRONG :=  AI_List_1[92 ],	WORD_WEAK := AI_List_1[92 ], SIZE := 1, FIX := 0, SIGNED := 0, VAR_OUT	:= MesDataExd.MesData.Mes20kVCourNeutCuveDecltI1);
MW(WORD_STRONG :=  AI_List_1[95 ],	WORD_WEAK := AI_List_1[95 ], SIZE := 1, FIX := 0, SIGNED := 0, VAR_OUT	:= MesDataExd.MesData.Mes20kVCourNeutCuveDecltI2);

MW(WORD_STRONG :=  AI_List_1[97  ],	WORD_WEAK := AI_List_1[97  ], SIZE := 1, FIX := 0, SIGNED := 0, VAR_OUT	:= MesDataExd.MesData.Mes20kVGeneralSepamI1);
MW(WORD_STRONG :=  AI_List_1[98  ],	WORD_WEAK := AI_List_1[98  ], SIZE := 1, FIX := 0, SIGNED := 0, VAR_OUT	:= MesDataExd.MesData.Mes20kVGeneralSepamI2);
MW(WORD_STRONG :=  AI_List_1[99  ],	WORD_WEAK := AI_List_1[99  ], SIZE := 1, FIX := 0, SIGNED := 0, VAR_OUT	:= MesDataExd.MesData.Mes20kVGeneralSepamI3);
MW(WORD_STRONG :=  AI_List_1[108 ],	WORD_WEAK := AI_List_1[108 ], SIZE := 1, FIX := 3, SIGNED := 0, VAR_OUT	:= MesDataExd.MesData.Mes20kVGeneralSepamU21);
MW(WORD_STRONG :=  AI_List_1[109 ],	WORD_WEAK := AI_List_1[109 ], SIZE := 1, FIX := 3, SIGNED := 0, VAR_OUT	:= MesDataExd.MesData.Mes20kVGeneralSepamU32);
MW(WORD_STRONG :=  AI_List_1[110 ],	WORD_WEAK := AI_List_1[110 ], SIZE := 1, FIX := 3, SIGNED := 0, VAR_OUT	:= MesDataExd.MesData.Mes20kVGeneralSepamU13);
MW(WORD_STRONG :=  AI_List_1[114 ],	WORD_WEAK := AI_List_1[114 ], SIZE := 1, FIX := 0, SIGNED := 0, VAR_OUT	:= MesDataExd.MesData.Mes20kVGeneralSepamResidualU);
MW(WORD_STRONG :=  AI_List_1[117 ],	WORD_WEAK := AI_List_1[117 ], SIZE := 1, FIX := 0, SIGNED := 0, VAR_OUT	:= MesDataExd.MesData.Mes20kVGeneralSepamFrequency);
MW(WORD_STRONG :=  AI_List_1[119 ],	WORD_WEAK := AI_List_1[119 ], SIZE := 1, FIX := 0, SIGNED := 0, VAR_OUT	:= MesDataExd.MesData.Mes20kVGeneralSepamP);
MW(WORD_STRONG :=  AI_List_1[120 ],	WORD_WEAK := AI_List_1[120 ], SIZE := 1, FIX := 0, SIGNED := 0, VAR_OUT	:= MesDataExd.MesData.Mes20kVGeneralSepamQ);
MW(WORD_STRONG :=  AI_List_1[123 ],	WORD_WEAK := AI_List_1[123 ], SIZE := 1, FIX := 0, SIGNED := 0, VAR_OUT	:= MesDataExd.MesData.Mes20kVGeneralSepamCosPhi);

MW(WORD_STRONG :=  AI_List_2[1 	 ], WORD_WEAK := AI_List_2[1 ], SIZE := 1, FIX := 0, SIGNED := 0, VAR_OUT	:= MesDataExd.MesData.Mes20kVMidiSepamI1);
MW(WORD_STRONG :=  AI_List_2[2   ], WORD_WEAK := AI_List_2[2 ], SIZE := 1, FIX := 0, SIGNED := 0, VAR_OUT	:= MesDataExd.MesData.Mes20kVMidiSepamI2);
MW(WORD_STRONG :=  AI_List_2[3   ], WORD_WEAK := AI_List_2[3 ], SIZE := 1, FIX := 0, SIGNED := 0, VAR_OUT	:= MesDataExd.MesData.Mes20kVMidiSepamI3);
MW(WORD_STRONG :=  AI_List_2[22  ], WORD_WEAK := AI_List_2[22 ], SIZE := 1, FIX := 0, SIGNED := 0, VAR_OUT	:= MesDataExd.MesData.Mes20kVMidiSepamP);
MW(WORD_STRONG :=  AI_List_2[23  ], WORD_WEAK := AI_List_2[23 ], SIZE := 1, FIX := 0, SIGNED := 0, VAR_OUT	:= MesDataExd.MesData.Mes20kVMidiSepamQ);
                                                        
MW(WORD_STRONG :=  AI_List_2[33 ], WORD_WEAK := AI_List_2[33 ], SIZE := 1, FIX := 0, SIGNED := 0, VAR_OUT	:= MesDataExd.MesData.Mes20kVPlatSepamI1);
MW(WORD_STRONG :=  AI_List_2[34 ], WORD_WEAK := AI_List_2[34 ], SIZE := 1, FIX := 0, SIGNED := 0, VAR_OUT	:= MesDataExd.MesData.Mes20kVPlatSepamI2);
MW(WORD_STRONG :=  AI_List_2[35 ], WORD_WEAK := AI_List_2[35 ], SIZE := 1, FIX := 0, SIGNED := 0, VAR_OUT	:= MesDataExd.MesData.Mes20kVPlatSepamI3);
MW(WORD_STRONG :=  AI_List_2[54 ], WORD_WEAK := AI_List_2[54 ], SIZE := 1, FIX := 0, SIGNED := 0, VAR_OUT	:= MesDataExd.MesData.Mes20kVPlatSepamP);
MW(WORD_STRONG :=  AI_List_2[55 ], WORD_WEAK := AI_List_2[55 ], SIZE := 1, FIX := 0, SIGNED := 0, VAR_OUT	:= MesDataExd.MesData.Mes20kVPlatSepamQ);

MW(WORD_STRONG :=  AI_List_2[97 ], WORD_WEAK := AI_List_2[97 ], SIZE := 1, FIX := 0, SIGNED := 0, VAR_OUT	:= MesDataExd.MesData.Mes20kVPlatSepamQ);


*)
END_METHOD

END_FUNCTION_BLOCK

// ---- 01_Equipement_Library/PCS/FB_PCS.TcPOU
FUNCTION_BLOCK FB_PCS EXTENDS FB_PCS_Base
//////////////////
// PLC controller . Jema Object 
//////////////////

VAR_INPUT PERSISTENT
	// Parameters of the Object
		ParamPnom							: REAL := 1500.0;	// (kW) Nominal power
		ParamQnom							: REAL := 1500.0;	// (kW) Nominal power
		ParamSmax							: REAL := 1500.0;	// (kVA) Maximum apparent power of the PCS (lasts 30s)
		
		ParamTimeoutCmdQ					: TIME := T#15S; 	// Time to activate or deactivate Q regulation before an alarm is raised
		ParamTimeoutCmdCosPhi				: TIME := T#15S; 	// Time to activate or deactivate CosPhi regulation before an alarm is raised
		ParamTimeoutQvU						: TIME := T#15S;	// Time to activate or deactivate Q(U) regulation before an alarm is raised
		ParamTimeoutPvF						: TIME := T#15S;	// Time to activate or deactivate P(f) regulation before an alarm is raised
    	                            		
		ParamSetPtModbusMode				: BOOL := TRUE;		// If True, then Setpoints come from Modbus
		ParamPoverQ							: BOOL := TRUE;		// If P over Q is True, then Max setpoint for Q calculated from setpoint of P
    	                    			
		ParamQfU_UDbHigh    				: REAL;				// JEMA U1 : AKUO U_UDbHigh
		ParamQfU_Umax		    			: REAL;				// JEMA U2 : AKUO U_Umax
		ParamQfU_UDbLow	    				: REAL;				// JEMA U3 : AKUO U_UDbLow
		ParamQfU_Umin		    			: REAL;				// JEMA U4 : AKUO U_Umin
		                            		
		ParamQfU_QDbHigh					: REAL;				// JEMA Q1 : AKUO U_QDbHigh
		ParamQfU_Qmax						: REAL;				// JEMA Q2 : AKUO U_Qmax
		ParamQfU_QDbLow						: REAL;				// JEMA Q3 : AKUO U_QDbLow
		ParamQfU_Qmin						: REAL;				// JEMA Q4 : AKUO U_Qmin
    	                            		
		ParamPfF_FDbHigh	    			: REAL;				// JEMA f1 : AKUO P_FDbHigh
		ParamPfF_Fmax		    			: REAL;				// JEMA f2 : AKUO P_Fmax
		ParamPfF_FDbLow	    				: REAL;				// JEMA f3 : AKUO P_FDbLow
		ParamPfF_Fmin		    			: REAL;				// JEMA f4 : AKUO P_Fmin
		                            		
		ParamPfF_PDbHigh					: REAL;				// JEMA P1 : AKUO P_PDbHigh
		ParamPfF_Pmax						: REAL;				// JEMA P2 : AKUO P_Pmax
		ParamPfF_PDbLow						: REAL;				// JEMA P3 : AKUO P_PDbLow
		ParamPfF_Pmin						: REAL;				// JEMA P4 : AKUO P_Pmin
    	
		ParamPfF_FhystLow					: REAL;				// JEMA fst1
		ParamPfF_FhystHigh					: REAL;				// JEMA fst2
		
		ParamFLow_droop						: REAL;				// (Hz) flow frequency (droop curve)
		ParamFHigh_droop					: REAL;				// (Hz) fhigh frequency (droop curve)
		ParamULow_droop						: REAL;				// (V) Ulow voltage (droop curve)
		ParamUHigh_droop					: REAL;				// (V) Ulow voltage (droop curve)
		
    	         	    		
		ParamTimeSoCRangeReachedRmp			: TIME;				// (ms) Time to ramp P back to the setpoint after the SoC reached its limits
		ParamTimeFreqRegStbDuration			: TIME;				// (ms) Time to ramp P back to the setpoint after entering the stable 
		ParamTimeEnterStblPriorRmp			: TIME; 			// (ms) Time to wait after entering the stable before ramping the P back to the setpoint
		    
    	                            	
		ParamTimeoutGridFormerTransition	: TIME := T#1M ;	// (ms) Time elapsed after grid former cmd when an alarm is raised
		ParamTimeoutGridFeederTransition	: TIME := T#1M;		// (ms) Time elapsed after grid feeder cmd when an alarm is raised
 		ParamTimeoutOffTransition			: TIME := T#1M;		// (ms) Time elapsed after CmdStop cmd when an alarm is raised
   	
		ParamFreqRegSoCmax 					: REAL;	 			// Jema Stops charging setpoint and overfreq regulation if BESS reaches this value
		ParamFreqRegSoCmin 					: REAL;				// Jema Stops discharging setpoint and underfreq regulation if BESS reaches this value
    	
		ParamLVRT_Enabled					: BOOL; 			// LVRT Enabled 
		ParamAntiIslanding_Enabled			: BOOL;				// Is Anti Islanding enabled

		ParamDeactivateWatchdog				: BOOL := TRUE;				// Parameter to deactivate the watchdog
		ParamMicroCyclingPower				: REAL;				// (kW) Active power the PCS will have during microcyling
		ParamMicroCyclingSoCMax				: REAL;				// (%) MaxSoC to reach before inverting Power
		ParamMicroCyclingSoCMin				: REAL;				// (%) MinSoC to reach before inverting Power
		ParamSocMax_L						: REAL;				// (%)  Max SOC Local
		ParamSocMin_L						: REAL;				// (%)  Min SOC Local
		ParamSocVeryVeryHigh				: REAL;				// (%) High SoC High Hysteresis
		ParamSocVeryHigh					: REAL;				// (%) High SoC Low Hysteresis
		ParamSocVeryVeryLow					: REAL;				// (%) Low SoC High Hysteresis
		ParamSocVeryLow						: REAL;				// (%) Low SoC Low Hysteresis 
				
 
	// Not Used at the moment : used to calculate theoretical Efficiency
		ParamRendementPcsNom				: REAL := 98;		// (%) Nominal Efficiency of the PCS at optimal conditions  
		ParamRendementPcsMin				: REAL := 80;		// (%) Minimal Efficiency of the PCS at P = 0  
		ParamTauxDeChargeRef				: REAL := 10;		// (%) LoadFactor where 1/5 of the efficiency is reached             			
END_VAR 
VAR_INPUT   	                   			
	// Commands :
		IN_CmdInvLocal						: BOOL;				// PCS is not included in available PCS' pool (excluded from HPP control). 
		IN_CmdStopOperation					: BOOL;				// BESS Specific command : Stop operation		
		IN_CmdPreventStart					: BOOL;				// BESS Specific command : Prevent start	
		IN_CmdOpenAC						: BOOL;				// Cmd To send an Open AC order
		IN_CmdOpenDC						: BOOL;				// Cmd To send an Open DC order	
 		IN_CmdP_On							: BOOL;				// Cmd start regulating on SetptP from outside of PCS : if you wan to know from what source, add a _IO2 value
		IN_CmdQ_On							: BOOL;				// Cmd start regulating on SetptQ from outside of PCS : if you wan to know from what source, add a _IO2 value
		IN_CmdCosPhi_On						: BOOL;				// Cmd start regulating on SetptCosPhi from outside of PCS : if you wan to know from what source, add a _IO2 value
		IN_CmdP_Off							: BOOL;				// Cmd start regulating on SetptP from outside of PCS : if you wan to know from what source, add a _IO2 value
		IN_CmdQ_Off							: BOOL;				// Cmd start regulating on SetptQ from outside of PCS : if you wan to know from what source, add a _IO2 value
		IN_CmdCosPhi_Off					: BOOL;				// Cmd start regulating on SetptCosPhi from outside of PCS : if you wan to know from what source, add a _IO2 value
		IN_CmdFreqregOn						: BOOL;				// Cmd 
		IN_CmdFreqregOff					: BOOL;				// 
		IN_CmdUregOn						: BOOL;				// 
		IN_CmdUregOff						: BOOL;				// 
		IN_CmdMicroCyclingOn				: BOOL;				// 
		IN_CmdMicroCyclingOff				: BOOL;				// 
		IN_CmdStandby						: BOOL;				// Cmd To send a soft Stop (No opening and closing of the AC/DC switch )
		IN_CmdStart							: BOOL;				// Cmd To send a start to the PCS (Does the full procedure, Soft + Close AC + Close DC)
		IN_CmdStop							: BOOL;				// Cmd To send a stop to the PCS (Soft Stop + Open DC + Open AC)
		
		                            		
		IN_CmdBlackStart					: BOOL; 			// Cmd Black start from outside of PCS : if you wan to know from what source, add a _IO2 value
		IN_CmdGridFormer					: BOOL;				// 
		IN_CmdGridFeeder					: BOOL;				// 
		IN_SetptP_Local						: REAL;				// Local Command
		IN_SetptQ_Local						: REAL;				// Local Command
		IN_SetptU_Local						: REAL := 500;	// Local Command
		IN_SetptF_Local						: REAL := 50;		// Local Command
		
		IN_CmdWatchdog						: BOOL ; 			// Activate or Deactivate the Watchdog function
	                
END_VAR
VAR_OUTPUT
	//Child objects
		OUT_SetptP_IO					: INT;			// (NA) Analogical value for the active power setpoint (based on ParamPnom)
		OUT_SetptQ_IO					: INT;			// (NA) Analogical value for the reactive power setpoint (based on ParamQnom)

END_VAR
VAR          


	MesDataExd								: PCS_Jema ;
                           	
	//M_ALARMMANAGEMENT VARIABLES//  
		AX_AlarmWords						: ARRAY[1..30] OF ST_ValuesAlarms;
		AX_AlarmWords_Null					: ARRAY[1..30] OF ST_ValuesAlarms;
		AX_AlarmWordsJema					: ARRAY[1..225] OF ST_ValuesAlarms;
		AX_AlarmWordsJema_Null				: ARRAY[1..225] OF ST_ValuesAlarms;
		NumAlarmsActive						: UINT;
		NumAlarmsActiveJema					: UINT;
	//M_READ VARIABLES//            		
		ModbusRead            				: ARRAY [1..4] OF FB_ModbusRead ; 	// (NA) FB for Modbus Reading
		MesBlock1_Temp						: ARRAY [1..4] OF ARRAY[1..120] OF WORD ; // (NA) Temporary Block Matrix for PCS modbus reading		
		AX_PcsHeartbit						: ARRAY [1..4] OF BOOL;
		                                	
		MesModbusReadAlarm 		  			: ARRAY [1..4] OF BOOL ;				// (NA) Modbus Read Alarm for communication
		TON_PcsHeartBitAlarm				: ARRAY [1..4] OF TON ;	
		TON_AlarmPcs						: ARRAY [1..4] OF TON ; 			// DesInhibate undervoltage alarms on PCS few seconds after PCS connected .  
                                        	
		DFV									: ARRAY[1..3] OF FB_DetectFixedValue;	
		StaticValuesToCompareHeartbit		: ARRAY[1..3] OF REAL;
		                                	                                     
		CTU_PcsNb							: CTU ; 
	

	// M_EVALUATE VARIABLES//
		DataHPP								: PP;
		DataPDL								: SUBMV_Exd;
		DataSystemBMS						: BAT;
		MesStatusWatchdog					: BOOL;
		MesHeartbeat_Old					: WORD;
		Trig_Watchdog						: R_TRIG;
		
	// Microcycling //
		MesMicroCyclingP					: REAL;				// (kW) Actual P for microcyling mode (if micro act = either ParamPmicro/-ParamPmicor, else 0)		
		MesMicroCyclingP_Old				: REAL;				// (kW) Active power the PCS will have during microcyling
	    MesMicroCyclingAllowed				: BOOL;				// (NA) If SoC is in range for microCycling                        		
		Trig_MicroCyclingNoLongerAllowed	: F_TRIG;			// Trig to detect falling edge of microcylingAllowed

	//M_WRITECOMMAND VARIABLES//    		
		ModbusWrite							: ARRAY [1..3] OF FB_ModbusWrite ;				// (NA) Functionnal Block for Writing Command Word through modbus
		Trig_Write							: ARRAY [1..3] OF R_TRIG;               		
		MesModbusWriteCmdAlarm				: ARRAY [1..3] OF BOOL ;						// (NA) Modbus Write Failed  (Command word) . 	
		MesModbusWriteCode          		: ARRAY [1..3] OF UDINT ; 						// (NA) Modbus Write Alarm Code 
		CmdWrite			AT%Q*			: ARRAY [1..3] OF BOOL;                     	
		AX_Cmd				AT%Q*			: ARRAY [1..3] OF ARRAY [1..120] OF WORD;   	
		AX_Cmd_Old							: ARRAY [1..3] OF ARRAY [1..120] OF WORD;   	
                                   		                                                	
		TRIG_CmdOpenAC						: R_TRIG;										// Trig to detect an order to change Mode
		TRIG_CmdOpenDC						: R_TRIG;										// Trig to detect an order to change Mode
		TRIG_CmdP_On						: R_TRIG;										// Trig to detect an order to change Mode
		TRIG_CmdQ_On			    		: R_TRIG;										// Trig to detect an order to change Mode
		TRIG_CmdCosPhi_On 					: R_TRIG;										// Trig to detect an order to change Mode
		TRIG_CmdP_Off						: R_TRIG;										// Trig to detect an order to change Mode
		TRIG_CmdQ_Off			    		: R_TRIG;										// Trig to detect an order to change Mode
		TRIG_CmdCosPhi_Off 					: R_TRIG;										// Trig to detect an order to change Mode
		TRIG_CmdBlackStart					: R_TRIG;										// Trig to detect an order to change Mode
		TRIG_CmdReset						: R_TRIG;		
		TRIG_FreqReg_On						: R_TRIG;
		TRIG_FreqReg_Off					: R_TRIG;
		TRIG_UReg_On						: R_TRIG;
		TRIG_UReg_Off						: R_TRIG;
		TRIG_CmdGridFormer					: R_TRIG;
		TRIG_CmdGridFeeder					: R_TRIG;
		TRIG_CmdMicroCyclingOn				: R_TRIG;
		TRIG_CmdMicroCyclingOff     		: R_TRIG;
		TRIG_CmdStop						: R_TRIG;
		TRIG_CmdStandby						: R_TRIG;
		TRIG_CmdStart						: R_TRIG;
		TRIG_CmdPcsLocal					: R_TRIG;
		TRIG_LowLowSoC						: R_TRIG;
		                            		
		TP_CmdBlackStart					: TP;				// TP To ensure R trig is detected
		TP_Reset							: TP ; 				// (NA) Maintain Reset command for a certain time 
		TP_CmdStandby						: TP;				// TP To maintain a soft stop order

		// Pour la commande start, j'envoie une consigne pour fermer les contacteurs DC des batteries
		TP_CmdOpenAC						: TP;				// TP To ensure R trig is detected
		TP_CmdOpenDC						: TP;				// TP To ensure R trig is detected

		TP_CmdStart							: TP;				// TP To ensure R trig is detected
		TP_CmdPreStart						: TP;				// TP To send a close dc breaker order before sending start order
		F_TrigPreStart						: F_TRIG;			// failing edge to detect end of TP;
		
		// Pour la commande stop, pour éviter qu'on ouvre tout d'un coup, je faire un pré stop pendant 1,5s où j'envoie un autre de standby
		TP_CmdStop							: TP;				// TP To ensure R trig is detected
		TP_CmdPreStop						: TP;				// TP to send a soft stop before sending a stop 
		F_TrigPreStop						: F_TRIG;			// failing edge to detect end of TP;
		                            		
		TON_CmdP_On							: TON;			// Trig to detect an order to change Mode
		TON_CmdQ_On			    			: TON;			// Trig to detect an order to change Mode
		TON_CmdCosPhi_On 					: TON;			// Trig to detect an order to change Mode
		TON_CmdP_Off						: TON;			// Trig to detect an order to change Mode
		TON_CmdQ_Off			    		: TON;			// Trig to detect an order to change Mode
		TON_CmdCosPhi_Off 					: TON;			// Trig to detect an order to change Mode
		TON_CmdBlackStart					: TON;			// Trig to detect an order to change Mode
		TON_FreqReg_On						: TON;
		TON_FreqReg_Off						: TON;
		TON_UReg_On							: TON;
		TON_UReg_Off						: TON;
		TON_CmdGridFormer					: TON;
		TON_CmdGridFeeder					: TON;
		TON_CmdMicroCyclingOn				: TON;
		TON_CmdMicroCyclingOff     			: TON;
		TON_CmdStart			    		: TON;
		TON_CmdStop	                		: TON;
		TON_CmdStandby		        		: TON;

		RS_hystlimitmin						: RS;
		RS_hystlimitmax						: RS;
 		RS_hystlimitEnergyShifmin			: RS;
		RS_hystlimitEnergyShifmax			: RS;
		
		CalPmaxCorr_highSoC					: REAL;
		CalPminCorr_lowSoC					: REAL;
        	           	                            		
END_VAR

METHOD M_AlarmManagement
//////////////////
//  PCS Alarm Management 
/////////////////

VAR 
	// Method local variables (reinitialized at each cycle) 
	FB_AlarmCodeManager : FB_AlarmCodeManager ; 
	KK					: UINT;				// For Loop
	ComWarning			: BOOL;				// Aggregated Wcommunication warning
	ComAlarm			: BOOL;				// Aggregated communication Alarm
	
	CalAlarmPcsSynthesis: BOOL;
	LL					: UINT;
	ID_Journal			: UINT;
	WordTest			: WORD;
	MesNbMots			: UINT;
END_VAR
// COMMUNICATION //
	ComWarning 				:=  MesModbusReadAlarm[1] OR MesModbusReadAlarm[2] OR MesModbusReadAlarm[3] ;		
	ComAlarm				:=  MesModbusReadAlarm[1] AND MesModbusReadAlarm[2] AND MesModbusReadAlarm[3]  ;
		
	TON_ComAlarm(IN:= ComAlarm , PT:= ParamTempoComAlarm, Q=>MesComAlarm) ;	
	TON_ComWarning(IN := ComWarning, PT := ParamTempoComWarning, Q => MesComWarning);
MesDataExd.MesData.MesComAlarm		:= MesComAlarm ; 
MesDataExd.MesData.MesComWarning 	:= MesComWarning ; 
	

// PCS ALARM INHIBITION
FOR KK := 1 TO ParamNbPcs DO
	TON_AlarmPcs[KK](IN:=NOT CalState.0, PT:= T#5S ) ;
	IF NOT TON_AlarmPcs[KK].Q THEN 
	MesDataExd.MesData.AX_PowerCol[KK].MesRegAlarm0.4 := FALSE ; 
	MesDataExd.MesData.AX_PowerCol[KK].MesRegAlarm0.7 := FALSE ; 
	MesDataExd.MesData.AX_PowerCol[KK].MesRegAlarm0.9 := FALSE ; 
	MesDataExd.MesData.AX_PowerCol[KK].MesRegAlarm0.11 := FALSE ; 
	MesDataExd.MesData.AX_PowerCol[KK].MesRegAlarm0.13 := FALSE ;			
	END_IF
	
	DFV[KK](IN_Addr := ADR(MesDataExd.MesData.AX_PowerCol[KK].MesHeartbit), IN_EmptyStruct := ADR(StaticValuesToCompareHeartbit[KK]) , IN_Size := SIZEOF(MesDataExd.MesData.AX_PowerCol[KK].MesHeartbit), IN_Duration := T#10S, OUT_bStatic => AX_PcsHeartbit[KK] ) ; 
	
END_FOR	


// SYNTHESES ALARMES //
CalAlarmPcsSynthesis := MesDataExd.MesData.AX_PowerCol[1].MesRegAlarm0 > 0
OR MesDataExd.MesData.AX_PowerCol[2].MesRegAlarm0 > 0
OR MesDataExd.MesData.AX_PowerCol[3].MesRegAlarm0 > 0
OR MesDataExd.MesData.AX_PowerCol[1].MesRegAlarm1 > 0
OR MesDataExd.MesData.AX_PowerCol[2].MesRegAlarm1 > 0
OR MesDataExd.MesData.AX_PowerCol[3].MesRegAlarm1 > 0
OR MesDataExd.MesData.AX_PowerCol[1].MesRegAlarm2 > 0
OR MesDataExd.MesData.AX_PowerCol[2].MesRegAlarm2 > 0
OR MesDataExd.MesData.AX_PowerCol[3].MesRegAlarm2 > 0
OR MesDataExd.MesData.AX_PowerCol[1].MesRegAlarm3 > 0
OR MesDataExd.MesData.AX_PowerCol[2].MesRegAlarm3 > 0
OR MesDataExd.MesData.AX_PowerCol[3].MesRegAlarm3 > 0
OR MesDataExd.MesData.AX_PowerCol[1].MesRegAlarm4 > 0
OR MesDataExd.MesData.AX_PowerCol[2].MesRegAlarm4 > 0
OR MesDataExd.MesData.AX_PowerCol[3].MesRegAlarm4 > 0 ;


// AlarmCode		
	FB_AlarmCodeManager(
		bAlarm1		:= CalAlarmPcsSynthesis		,								// Power columns Alarm Synthesis, at least one alarm active on power column
		bAlarm2		:= TON_CmdP_On.Q OR TON_CmdP_Off.Q,							// Timeout for CmdP order
		bAlarm3		:= TON_CmdQ_On.Q OR TON_CmdQ_Off.Q,							// Timeout for CmdQ order			
		bAlarm4		:= FALSE,										            //                              			    	
		bAlarm5		:= TON_CmdBlackStart.Q,                                     // Timeout for BlackStart order   			
		bAlarm6		:= TON_FreqReg_On.Q OR TON_FreqReg_Off.Q,                   // Timeout for Freq Regulation activation                            				
		bAlarm7		:= TON_UReg_On.Q OR TON_UReg_Off.Q,                         // Timeout for Voltage Regulation activation
		bAlarm8 	:= TON_CmdGridFormer.Q,                                     // Timeout for grid former activation
		bAlarm9		:= TON_CmdGridFeeder.Q,                                     // Timeout for grid feeder activation
		bAlarm10	:= TON_CmdMicroCyclingOn.Q OR TON_CmdMicroCyclingOff.Q,     // Timeout for MicroCycling
		bAlarm11	:= MesDataExd.MesData.MesComAlarm,                                     // Communication alarm : none of the Power Columns are responding 				
		bAlarm12	:= FALSE,                                               	//				
		bAlarm13	:= FALSE,                                               	//			
		bAlarm14	:= FALSE,                                               	//		
		bAlarm15	:= FALSE,                                               	//		
		wAlarmCode	=>MesDataExd.MesData.MesAlarmCode);		                                		
		                                                                                 	
		
		
// WARNING CODE //
	FB_AlarmCodeManager(
		bAlarm1		:= MesComWarning, 																															// Communication warning : At least one of the Power Columns are not responding 
		bAlarm2		:= FALSE,																																	// 
		bAlarm3		:= MesDataExd.MesData.AX_PowerCol[1].MesDeratingWord.0  ,  																							// Power Column 1 derating active due to temperature
		bAlarm4		:= MesDataExd.MesData.AX_PowerCol[2].MesDeratingWord.0,    																							// Power Column 2 derating active due to temperature
		bAlarm5		:= MesDataExd.MesData.AX_PowerCol[3].MesDeratingWord.0,  																								// Power Column 3 derating active due to temperature
		bAlarm6		:= MesDataExd.MesData.AX_PowerCol[1].MesDeratingWord.4 OR MesDataExd.MesData.AX_PowerCol[2].MesDeratingWord.4 OR MesDataExd.MesData.AX_PowerCol[3].MesDeratingWord.4,      	// At least one power column has a derating due to overvoltage
		bAlarm7		:= MesDataExd.MesData.AX_PowerCol[1].MesDeratingWord.5 OR MesDataExd.MesData.AX_PowerCol[2].MesDeratingWord.5 OR MesDataExd.MesData.AX_PowerCol[3].MesDeratingWord.5,      	// At least one power column has a derating due to undervoltage
		bAlarm8		:= MesDataExd.MesData.AX_PowerCol[1].MesDeratingWord.6 OR MesDataExd.MesData.AX_PowerCol[2].MesDeratingWord.6 OR MesDataExd.MesData.AX_PowerCol[3].MesDeratingWord.6,      	// At least one power column has a derating due to overfrequency
		bAlarm9		:= MesDataExd.MesData.AX_PowerCol[1].MesDeratingWord.7 OR MesDataExd.MesData.AX_PowerCol[2].MesDeratingWord.7 OR MesDataExd.MesData.AX_PowerCol[3].MesDeratingWord.7,      	// At least one power column has a derating due to underfrequency
		bAlarm10	:= MesDataExd.MesData.AX_PowerCol[1].MesDoorOpened,           																							// Power column 1 cabinet door is opened
		bAlarm11	:= MesDataExd.MesData.AX_PowerCol[2].MesDoorOpened,           																							// Power column 2 cabinet door is opened
		bAlarm12	:= MesDataExd.MesData.AX_PowerCol[3].MesDoorOpened,           																							// Power column 3 cabinet door is opened
		bAlarm13	:= FALSE,           																														//
		bAlarm14	:= FALSE,           																														//
		bAlarm15	:= FALSE,           																														//
		wAlarmCode	=>MesDataExd.MesData.MesWarningCode);
		
// EVENT CODE //
	FB_AlarmCodeManager(
		bAlarm1			:= MesDataExd.MesData.AX_PowerCol[1].MesAcSwitchClosed,																							// AC Switch Closed for PCS 1
		bAlarm2			:= NOT MesDataExd.MesData.MesDcBreaker, 																											// DC Switch Closed
		bAlarm3			:= MesDataExd.MesData.OUT_CmdStandby, 																												// Soft stop command
		bAlarm4			:= MesDataExd.MesData.MesOnGrid,																													// OnGrid Mode is activated
		bAlarm5			:= MesDataExd.MesData.MesOffGrid, 																													// Offgrid Mode is activated
		bAlarm6			:= MesDataExd.MesData.OUT_CmdStart, 																												// Cmd Start
		bAlarm7			:= MesDataExd.MesData.OUT_CmdStop, 																												// Full stop command
		bAlarm8			:= MesDataExd.MesData.OUT_CmdBlackStart, 																											// Cmd BlackStart
		bAlarm9			:= MesDataExd.MesData.AX_PowerCol[1].MesRegAlarm2.9 OR MesDataExd.MesData.AX_PowerCol[2].MesRegAlarm2.9 OR MesDataExd.MesData.AX_PowerCol[3].MesRegAlarm2.9,			// Grid collapsed 
		bAlarm10		:= MesDataExd.MesData.AX_PowerCol[2].MesAcSwitchClosed,																							// AC Switch Closed for PCS 2
		bAlarm11		:= SEL(ParamNbPcs>2 ,  FALSE, MesDataExd.MesData.AX_PowerCol[3].MesAcSwitchClosed),																// AC Switch Closed for PCS 3
		bAlarm12		:= NOT MesDataExd.MesData.MesAcBreaker, 																											// Ac breaker is Closed. 
		bAlarm13		:= MesDataExd.MesData.MesPrecharge,                                                                                            					// ESS - INV : Precharge
		bAlarm14		:= NOT MesDataExd.MesData.OUT_CmdGridMode,                                                                                                         // OnGrid command
		bAlarm15		:= MesDataExd.MesData.OUT_CmdGridMode, 																											// OffGrid command
		wAlarmCode		=>MesDataExd.MesData.MesEventCode);                                                                                           					// 
		

NumAlarmsActive := 0;
AX_AlarmWords := AX_AlarmWords_Null;
MesNbMots := 2;
FOR KK := 1 TO MesNbMots DO			// Combien j'ai de mots
	ID_Journal := 15 + (ParamEssNum-1) * MesNbMots * CstNbPcs_ESS_G + (ParamPcsNum - 1) * CstNbPcs_ESS_G + (KK- 1);
	FOR LL := 1 TO 15 DO 	// Les bits 
		WordTest := ROR(FUN_Alarms.AX_RecupWord[ID_Journal],LL);
		IF WordTest.0 THEN
			NumAlarmsActive := NumAlarmsActive + 1;
			AX_AlarmWords[NumAlarmsActive].Message := FUN_Alarms.AX_Journal[ID_Journal][LL].Message;
		ELSE
			AX_AlarmWords[NumAlarmsActive+1].Message := '';
		END_IF
	END_FOR
END_FOR		

NumAlarmsActiveJema := 0;
AX_AlarmWordsJema := AX_AlarmWordsJema_Null;
MesNbMots := 15;
FOR KK := 1 TO MesNbMots DO			// Combien j'ai de mots
	FOR LL := 1 TO 15 DO 	// Les bits 
		ID_Journal := 57 + (ParamEssNum-1) * MesNbMots * CstNbPcs_ESS_G + (ParamPcsNum - 1) * CstNbPcs_ESS_G + (KK- 1);
		WordTest := ROR(FUN_Alarms.AX_RecupWord[ID_Journal],LL);
		IF WordTest.0 THEN
			NumAlarmsActiveJema := NumAlarmsActiveJema + 1;
			AX_AlarmWordsJema[NumAlarmsActiveJema].Message := FUN_Alarms.AX_Journal[ID_Journal][LL].Message;
		ELSE
			AX_AlarmWordsJema[NumAlarmsActiveJema+1].Message := '';
		END_IF
	END_FOR
END_FOR
END_METHOD

METHOD M_CP
//////////////////
//  Emulator
/////////////////

VAR 
	// Method local variables (reinitialized at each cycle) 
	
END_VAR
SUPER^.M_CP();
END_METHOD

METHOD M_Evaluate : BOOL
VAR_INPUT
END_VAR
VAR
	KK : UINT;
	bTest: BOOL;
	MesAlarmPcs: BOOL;
	AX_Journal : ARRAY[57..57] of array[1..15] of ST_ValuesAlarms;
END_VAR

// External values update :
DataHPP			:= A1_PP.MesDataExd.MesData.
DataSystemBMS 	:= AX_ESS[ParamEssNum].AX_BAT[ParamPcsNum].MesDataExd.MesData.
DataPDL 		:= A1_SUBMV.MesDataExd.MesData.

Trig_Watchdog(CLK := MesHeartbeat_Old <>MesDataExd.MesData.MesHeartBeat);
IF Trig_Watchdog.Q 	THEN
	MesHeartbeat_Old := MesDataExd.MesData.MesHeartBeat;
	MesStatusWatchdog := NOT MesStatusWatchdog;
END_IF

// PROPERTIES UPDATE // 
	// Controller
MesDataExd.MesData.MesP 	:= 0 ; 
MesDataExd.MesData.MesPdc 	:= 0 ;
MesDataExd.MesData.MesQ 	:= 0 ; 
MesDataExd.MesData.MesI 	:= 0 ; 			
MesDataExd.MesData.MesIdc 	:= 0 ; 		


MesDataExd.MesData.MesComAlarm					:= TRUE ; 						// All PCS in Com alarm . 			
MesDataExd.MesData.MesAtLeastOnePcsConnected 	:= FALSE  ; 	// At least one inverter connected and not in alarm			
MesDataExd.MesData.MesFreqReg_Active 			:= FALSE;
MesDataExd.MesData.MesUReg_Active 				:= FALSE;

	// Update PCS Values	
	FOR KK:= 1 TO ParamNbPcs DO 
	MesDataExd.MesData.MesP 						:= MesDataExd.MesData.AX_PowerCol[KK].MesP + MesDataExd.MesData.MesP  ; 
	MesDataExd.MesData.MesI 						:= MesDataExd.MesData.AX_PowerCol[KK].MesI + MesDataExd.MesData.MesI  ; 
	MesDataExd.MesData.MesPdc 						:= MesDataExd.MesData.AX_PowerCol[KK].MesPdc + MesDataExd.MesData.MesPdc  ; 
		// ATTENTION MODIF RELATIVE A JEMA, JE METS UN MOINS PSK ILS SONT CONS
	MesDataExd.MesData.MesQ 						:= -.MesDataExd.MesData.AX_PowerCol[KK].MesQ + MesDataExd.MesData.MesQ  ; 
	MesDataExd.MesData.MesIdc 						:= MesDataExd.MesData.AX_PowerCol[KK].MesIdc + MesDataExd.MesData.MesIdc  ; 
	MesDataExd.MesData.MesFreqReg_Active			:= MesDataExd.MesData.MesFreqReg_Active 			OR MesDataExd.MesData.AX_PowerCol[KK].MesDeratingWord.6 OR MesDataExd.MesData.AX_PowerCol[KK].MesDeratingWord.7 ;
	MesDataExd.MesData.MesUReg_Active				:= MesDataExd.MesData.MesUReg_Active 				OR MesDataExd.MesData.AX_PowerCol[KK].MesDeratingWord.4 OR MesDataExd.MesData.AX_PowerCol[KK].MesDeratingWord.5 ;
		MesAlarmPcs							:= MesDataExd.MesData.AX_PowerCol[KK].MesRegAlarm0 > 0 OR MesDataExd.MesData.AX_PowerCol[KK].MesRegAlarm1 > 0 	OR MesDataExd.MesData.AX_PowerCol[KK].MesRegAlarm2 > 0 OR MesDataExd.MesData.AX_PowerCol[KK].MesRegAlarm3 > 0 OR MesDataExd.MesData.AX_PowerCol[KK].MesRegAlarm4 > 0);                                        	
	MesDataExd.MesData.MesComAlarm					:= MesDataExd.MesData.MesComAlarm 					AND AX_PcsHeartbit[KK];
	MesDataExd.MesData.MesAtLeastOnePcsConnected 	:= MesDataExd.MesData.MesAtLeastOnePcsConnected 	OR MesDataExd.MesData.AX_PowerCol[KK].MesAcSwitchClosed (*FAT TESTAND NOT MesAlarmPcs *);
		


		
	MesDataExd.MesData.AX_PowerCol[KK].MesJemaAlarms.MesI1_Alm					:= MesDataExd.MesData.AX_PowerCol[KK].MesRegAlarm0.0;
	MesDataExd.MesData.AX_PowerCol[KK].MesJemaAlarms.MesI2_Alm					:= MesDataExd.MesData.AX_PowerCol[KK].MesRegAlarm0.1;
	MesDataExd.MesData.AX_PowerCol[KK].MesJemaAlarms.MesI3_Alm					:= MesDataExd.MesData.AX_PowerCol[KK].MesRegAlarm0.2;
	MesDataExd.MesData.AX_PowerCol[KK].MesJemaAlarms.MesVdc_High_Alm			:= MesDataExd.MesData.AX_PowerCol[KK].MesRegAlarm0.3;
	MesDataExd.MesData.AX_PowerCol[KK].MesJemaAlarms.MesVdc_Low_Alm			:= MesDataExd.MesData.AX_PowerCol[KK].MesRegAlarm0.4;
	MesDataExd.MesData.AX_PowerCol[KK].MesJemaAlarms.MesU12_High_Alm			:= MesDataExd.MesData.AX_PowerCol[KK].MesRegAlarm0.6;
	MesDataExd.MesData.AX_PowerCol[KK].MesJemaAlarms.MesU12_Low_Alm			:= MesDataExd.MesData.AX_PowerCol[KK].MesRegAlarm0.7;
	MesDataExd.MesData.AX_PowerCol[KK].MesJemaAlarms.MesU23_High_Alm			:= MesDataExd.MesData.AX_PowerCol[KK].MesRegAlarm0.8;
	MesDataExd.MesData.AX_PowerCol[KK].MesJemaAlarms.MesU23_Low_Alm	 		:= MesDataExd.MesData.AX_PowerCol[KK].MesRegAlarm0.9;
	MesDataExd.MesData.AX_PowerCol[KK].MesJemaAlarms.MesU31_High_Alm			:= MesDataExd.MesData.AX_PowerCol[KK].MesRegAlarm0.10;
	MesDataExd.MesData.AX_PowerCol[KK].MesJemaAlarms.MesU31_Low_Alm	 		:= MesDataExd.MesData.AX_PowerCol[KK].MesRegAlarm0.11;
	MesDataExd.MesData.AX_PowerCol[KK].MesJemaAlarms.MesVd_High_Alm			:= MesDataExd.MesData.AX_PowerCol[KK].MesRegAlarm0.12;
	MesDataExd.MesData.AX_PowerCol[KK].MesJemaAlarms.MesVd_Low_Alm				:= MesDataExd.MesData.AX_PowerCol[KK].MesRegAlarm0.13;
	MesDataExd.MesData.AX_PowerCol[KK].MesJemaAlarms.MesVdc_Neg				:= MesDataExd.MesData.AX_PowerCol[KK].MesRegAlarm0.14;
	MesDataExd.MesData.AX_PowerCol[KK].MesjemaAlarms.MesU1223_Unbalance		:= MesDataExd.MesData.AX_PowerCol[KK].MesRegAlarm1.0;
	MesDataExd.MesData.AX_PowerCol[KK].MesjemaAlarms.MesU2331_Unbalance		:= MesDataExd.MesData.AX_PowerCol[KK].MesRegAlarm1.1;
	MesDataExd.MesData.AX_PowerCol[KK].MesjemaAlarms.MesU3112_Unbalance		:= MesDataExd.MesData.AX_PowerCol[KK].MesRegAlarm1.2;
	MesDataExd.MesData.AX_PowerCol[KK].MesjemaAlarms.MesInvertedPhase			:= MesDataExd.MesData.AX_PowerCol[KK].MesRegAlarm1.3;
	MesDataExd.MesData.AX_PowerCol[KK].MesjemaAlarms.MesI12_Unbalance			:= MesDataExd.MesData.AX_PowerCol[KK].MesRegAlarm1.4;
	MesDataExd.MesData.AX_PowerCol[KK].MesjemaAlarms.MesI23_Unbalance			:= MesDataExd.MesData.AX_PowerCol[KK].MesRegAlarm1.5;
	MesDataExd.MesData.AX_PowerCol[KK].MesjemaAlarms.MesI31_Unbalance			:= MesDataExd.MesData.AX_PowerCol[KK].MesRegAlarm1.6;
	MesDataExd.MesData.AX_PowerCol[KK].MesjemaAlarms.MesCouplingTimeout		:= MesDataExd.MesData.AX_PowerCol[KK].MesRegAlarm1.7;
	MesDataExd.MesData.AX_PowerCol[KK].MesjemaAlarms.MesF_High					:= MesDataExd.MesData.AX_PowerCol[KK].MesRegAlarm1.8;
	MesDataExd.MesData.AX_PowerCol[KK].MesjemaAlarms.MesF_Low			 		:= MesDataExd.MesData.AX_PowerCol[KK].MesRegAlarm1.9;
	MesDataExd.MesData.AX_PowerCol[KK].MesjemaAlarms.MesGrndFault				:= MesDataExd.MesData.AX_PowerCol[KK].MesRegAlarm1.10;
	MesDataExd.MesData.AX_PowerCol[KK].MesjemaAlarms.MesVaristor		 		:= MesDataExd.MesData.AX_PowerCol[KK].MesRegAlarm1.11;
	MesDataExd.MesData.AX_PowerCol[KK].MesjemaAlarms.MesPcbOverTemp			:= MesDataExd.MesData.AX_PowerCol[KK].MesRegAlarm1.12;
	MesDataExd.MesData.AX_PowerCol[KK].MesjemaAlarms.MesHeatsinkOverTemp		:= MesDataExd.MesData.AX_PowerCol[KK].MesRegAlarm1.13;
	MesDataExd.MesData.AX_PowerCol[KK].MesjemaAlarms.MesOvertempHyst			:= MesDataExd.MesData.AX_PowerCol[KK].MesRegAlarm1.15;		
	MesDataExd.MesData.AX_PowerCol[KK].MesJemaAlarms.MesGridCbOpened			:= MesDataExd.MesData.AX_PowerCol[KK].MesRegAlarm2.4;
	MesDataExd.MesData.AX_PowerCol[KK].MesJemaAlarms.MesGridCbTrip				:= MesDataExd.MesData.AX_PowerCol[KK].MesRegAlarm2.5;
	MesDataExd.MesData.AX_PowerCol[KK].MesJemaAlarms.MesGridContactFail		:= MesDataExd.MesData.AX_PowerCol[KK].MesRegAlarm2.8;
	MesDataExd.MesData.AX_PowerCol[KK].MesJemaAlarms.MesDoorOpened				:= MesDataExd.MesData.AX_PowerCol[KK].MesRegAlarm2.9;
	MesDataExd.MesData.AX_PowerCol[KK].MesJemaAlarms.MesVdcPrechargewrong		:= MesDataExd.MesData.AX_PowerCol[KK].MesRegAlarm2.12;
	MesDataExd.MesData.AX_PowerCol[KK].MesJemaAlarms.MesOverVoltHyst			:= MesDataExd.MesData.AX_PowerCol[KK].MesRegAlarm2.14;
	MesDataExd.MesData.AX_PowerCol[KK].MesJemaAlarms.MesIdcMax					:= MesDataExd.MesData.AX_PowerCol[KK].MesRegAlarm2.15;
	MesDataExd.MesData.AX_PowerCol[KK].MesjemaAlarms.MesSKIIP1					:= MesDataExd.MesData.AX_PowerCol[KK].MesRegAlarm3.0;
	MesDataExd.MesData.AX_PowerCol[KK].MesjemaAlarms.MesSKIIP2					:= MesDataExd.MesData.AX_PowerCol[KK].MesRegAlarm3.1;
	MesDataExd.MesData.AX_PowerCol[KK].MesjemaAlarms.MesSKIIP3					:= MesDataExd.MesData.AX_PowerCol[KK].MesRegAlarm3.2;
	MesDataExd.MesData.AX_PowerCol[KK].MesJemaAlarms.MesSKIIP_OT				:= MesDataExd.MesData.AX_PowerCol[KK].MesRegAlarm3.3;
	MesDataExd.MesData.AX_PowerCol[KK].MesjemaAlarms.MesIMax					:= MesDataExd.MesData.AX_PowerCol[KK].MesRegAlarm3.4;
	MesDataExd.MesData.AX_PowerCol[KK].MesjemaAlarms.MesEmergencyStop			:= MesDataExd.MesData.AX_PowerCol[KK].MesRegAlarm3.5;
	MesDataExd.MesData.AX_PowerCol[KK].MesjemaAlarms.MesFPGA_WdogTrip			:= MesDataExd.MesData.AX_PowerCol[KK].MesRegAlarm3.6;
	MesDataExd.MesData.AX_PowerCol[KK].MesjemaAlarms.MesStopEverything			:= MesDataExd.MesData.AX_PowerCol[KK].MesRegAlarm3.7;
	MesDataExd.MesData.AX_PowerCol[KK].MesjemaAlarms.MesImdWarning				:= MesDataExd.MesData.AX_PowerCol[KK].MesRegAlarm3.8;
	MesDataExd.MesData.AX_PowerCol[KK].MesjemaAlarms.MesImdFault				:= MesDataExd.MesData.AX_PowerCol[KK].MesRegAlarm3.9;
	MesDataExd.MesData.AX_PowerCol[KK].MesjemaAlarms.MesCoilOverTemp			:= MesDataExd.MesData.AX_PowerCol[KK].MesRegAlarm3.11;
	MesDataExd.MesData.AX_PowerCol[KK].MesjemaAlarms.MesAlrmGrp1_Curr			:= MesDataExd.MesData.AX_PowerCol[KK].MesRegAlarm3.13;
	MesDataExd.MesData.AX_PowerCol[KK].MesjemaAlarms.MesAlrmGrp2_Curr	 		:= MesDataExd.MesData.AX_PowerCol[KK].MesRegAlarm3.14;
	MesDataExd.MesData.AX_PowerCol[KK].MesjemaAlarms.MesShortCircuit_DC	 	:= MesDataExd.MesData.AX_PowerCol[KK].MesRegAlarm3.15;
	MesDataExd.MesData.AX_PowerCol[KK].MesjemaAlarms.MesBatError				:= MesDataExd.MesData.AX_PowerCol[KK].MesRegAlarm4.0;
	MesDataExd.MesData.AX_PowerCol[KK].MesjemaAlarms.MesBatCtlStop				:= MesDataExd.MesData.AX_PowerCol[KK].MesRegAlarm4.1;
	MesDataExd.MesData.AX_PowerCol[KK].MesjemaAlarms.MesBatComErrors			:= MesDataExd.MesData.AX_PowerCol[KK].MesRegAlarm4.2;
	MesDataExd.MesData.AX_PowerCol[KK].MesjemaAlarms.MesPowerUnbalance			:= MesDataExd.MesData.AX_PowerCol[KK].MesRegAlarm4.3;
	MesDataExd.MesData.AX_PowerCol[KK].MesjemaAlarms.MesOverpower				:= MesDataExd.MesData.AX_PowerCol[KK].MesRegAlarm4.4;

		
	END_FOR 
	
MesDataExd.MesData.MesCosPhi 				:= SEL(	MesDataExd.MesData.MesP=0) AND  MesDataExd.MesData.MesQ =0 ), MesDataExd.MesData.MesP / SQRT(EXPT.MesDataExd.MesData.MesP, 2) + EXPT.MesDataExd.MesData.MesQ, 2))   , 1) ; 		
MesDataExd.MesData.MesFreq					:= SEL.MesDataExd.MesData.AX_PowerCol[1].MesFreq=0 MesDataExd.MesData.AX_PowerCol[1].MesFreq , SEL.MesDataExd.MesData.AX_PowerCol[2].MesFreq=0 MesDataExd.MesData.AX_PowerCol[2].MesFreq MesDataExd.MesData.AX_PowerCol[3].MesFreq ))   ; 		
MesDataExd.MesData.MesU 					:= SEL.MesDataExd.MesData.AX_PowerCol[1].MesU=0 MesDataExd.MesData.AX_PowerCol[1].MesU , SEL.MesDataExd.MesData.AX_PowerCol[2].MesU=0 MesDataExd.MesData.AX_PowerCol[2].MesU MesDataExd.MesData.AX_PowerCol[3].MesU ))   ; 		
MesDataExd.MesData.MesUdc 					:= SEL.MesDataExd.MesData.AX_PowerCol[1].MesUdc=0 MesDataExd.MesData.AX_PowerCol[1].MesUdc , SEL.MesDataExd.MesData.AX_PowerCol[2].MesUdc=0 MesDataExd.MesData.AX_PowerCol[2].MesUdc MesDataExd.MesData.AX_PowerCol[3].MesUdc ))   ; 			
	 
//--------------------------------------------------------------------------------//
// 							Gestion des setpoints								  //
//--------------------------------------------------------------------------------//
	
// Gestion de la puissance dispo batterie		
	/  MesDataExd.MesData.CalDynamicEfficiencyPcs := (ParamRendementPcsNom  - ParamRendementPcsMin)* (1-EXP(-(abs.MesDataExd.MesData.CalP)/ParamPnom)*100/ParamTauxDeChargeRef)) + ParamRendementPcsMin;

// Gestion des limites hautes de SoC
	RS_hystlimitmax(SET:= DataSystemBMS.MesSoCConnected>= A1_PP.ParamSocMax_G , RESET1:= DataSystemBMS.MesSoCConnected< A1_PP.ParamSocVeryHigh) ; 
	RS_hystlimitmin(SET:= DataSystemBMS.MesSoCConnected<= A1_PP.ParamSocMin_G , RESET1:= DataSystemBMS.MesSoCConnected> A1_PP.ParamSocVeryLow) ; 
	
	IF DataSystemBMS.MesSoCConnected >= ParamSocVeryHigh THEN
		CalPmaxCorr_highSoC := (A1_PP.ParamSocMax_G - DataSystemBMS.MesSoCConnected)/(A1_PP.ParamSocMax_G - A1_PP.ParamSocVeryHigh );
	ELSE 
		CalPmaxCorr_highSoC := 1 ;
	END_IF 
	IF DataSystemBMS.MesSoCConnected <= ParamSocMin_L THEN
	CalPminCorr_lowSoC := (A1_PP.ParamSocMin_G - DataSystemBMS.MesSoCConnected)/(A1_PP.ParamSocMin_G - A1_PP.ParamSocVeryLow );
	ELSE
		CalPminCorr_lowSoC := 1;
	END_IF
	IF (datasystembms.MesCCL <> 0 OR datasystembms.MesDCL <> 0) AND DataSystemBMS.MesUdcConnected <> 0 THEN
	MesDataExd.MesData.MesS_BatChargeMax 		:=  SEL(RS_hystlimitmax.Q1, 1, 0) * CalPmaxCorr_highSoC * MIN(DataSystemBMS.MesCCL* DataSystemBMS.MesNbRackConnected,	ParamPnom);
	MesDataExd.MesData.MesS_BatDischargeMax 	:=  SEL(RS_hystlimitmin.Q1, 1, 0) * CalPminCorr_lowSoC * MIN(DataSystemBMS.MesDCL* DataSystemBMS.MesNbRackConnected,	ParamPnom);
	ELSE
	MesDataExd.MesData.MesS_BatChargeMax := 0;
	MesDataExd.MesData.MesS_BatDischargeMax := 0;
	END_IF

// Local
	// Si je suis en local, je désactive le micro cycling et je réecris le setpoint d'input	
	IF MesDataExd.MesData.OUT_CmdInvLocal THEN
	MesDataExd.MesData.OUT_CmdMicroCyclingMode := FALSE;
		IN_SetptP := IN_SetptP_Local;
		IN_SetptQ := IN_SetptQ_Local;
		IN_SetptU := IN_SetptU_Local;
		IN_SetptF := IN_SetptF_Local;
	END_IF

// MicroCycling
	// j'évalue si j'ai le droit de faire du micro-cycling
	MesMicroCyclingAllowed := DataSystemBMS.MesSoC >= ParamMicroCyclingSoCMin*0.95 AND DataSystemBMS.MesSoC <= ParamMicroCyclingSoCMax*1.05 ;
	Trig_MicroCyclingNoLongerAllowed(CLk := MesMicroCyclingAllowed);

	// Si je suis en mode micro cycling, dès que je passe au dessus du soc max, je décharge la batterie
	IF MesDataExd.MesData.OUT_CmdMicroCyclingMode AND DataSystemBMS.MesSoC >= ParamMicroCyclingSoCMax THEN
		IN_SetptP := ABS(ParamMicroCyclingPower);
	END_IF
	// Sinon, je la recharge
	IF MesDataExd.MesData.OUT_CmdMicroCyclingMode AND DataSystemBMS.MesSoC <= ParamMicroCyclingSoCMin THEN
		IN_SetptP := -ABS(ParamMicroCyclingPower);
	END_IF

	// et si je vois que la puissance de consigne change, je la réecris (en gardant le bon sens charge/décharge)
	IF MesMicroCyclingP_Old <> ParamMicroCyclingPower THEN
		MesMicroCyclingP_Old := ParamMicroCyclingPower;
		IN_SetptP := SEL(IN_SetptP > 0, -ABS(ParamMicroCyclingPower), ABS(ParamMicroCyclingPower));
	END_IF

IF ParamPoverQ THEN 
	// Le setpoint Max correspond à la dispo * la puissance nominale
MesDataExd.MesData.OUT_SetptPMax := MIN(MesDataExd.MesData.MesS_BatDischargeMax, MesDataExd.MesData.MesAvailability * MesDataExd.MesData.MesSnom/100.0,  SEL(DataSystemBMS.MesSoCConnected <= A1_PP.ParamSocMin_G, ParamPnom, 0));
MesDataExd.MesData.OUT_SetptPMin := MAX( MesDataExd.MesData.MesS_BatChargeMax, MesDataExd.MesData.MesAvailability * MesDataExd.MesData.MesSnom/100.0, SEL(DataSystemBMS.MesSoCConnected >= A1_PP.ParamSocMax_G, -ParamPnom, 0));

	// Min
	IF ABS.MesDataExd.MesData.MesS_BatDischargeMax) > ABS.MesDataExd.MesData.OUT_SetptP) THEN
	MesDataExd.MesData.OUT_SetptQMax		:= SQRT(EXPT.MesDataExd.MesData.MesS_BatDischargeMax, 2) - EXPT.MesDataExd.MesData.OUT_SetptP, 2));
	ELSE
	MesDataExd.MesData.OUT_SetptQMin := 0;
	END_IF
	IF ABS.MesDataExd.MesData.MesS_BatChargeMax) > ABS.MesDataExd.MesData.OUT_SetptP) THEN
	MesDataExd.MesData.OUT_SetptQMin		:= -SQRT(EXPT.MesDataExd.MesData.MesS_BatChargeMax, 2) - EXPT.MesDataExd.MesData.OUT_SetptP, 2));
	ELSE 
	MesDataExd.MesData.OUT_SetptQMin := 0;
	END_IF
ELSE
MesDataExd.MesData.OUT_SetptQMax := SEL.MesDataExd.MesData.MesP = 0, SEL.MesDataExd.MesData.MesP>0, MesDataExd.MesData.MesS_BatChargeMax, MesDataExd.MesData.MesS_BatDischargeMax), MIN(MesDataExd.MesData.MesS_BatChargeMax.MesDataExd.MesData.MesS_BatDischargeMax));
MesDataExd.MesData.OUT_SetptQMin := -.MesDataExd.MesData.OUT_SetptQMax;
	
MesDataExd.MesData.OUT_SetptPMax		:= MIN(SQRT(EXPT.MesDataExd.MesData.MesS_BatChargeMax, 2) - EXPT.MesDataExd.MesData.OUT_SetptQ, 2)),  SEL(DataSystemBMS.MesSoCConnected < A1_PP.ParamSocMin_G, ParamPnom, 0));
MesDataExd.MesData.OUT_SetptPMin		:= MAX(SQRT(EXPT.MesDataExd.MesData.MesS_BatDischargeMax, 2) - EXPT.MesDataExd.MesData.OUT_SetptQ, 2)),  SEL(DataSystemBMS.MesSoCConnected > A1_PP.ParamSocMax_G, ParamPnom, 0));
END_IF

// J'affecte les variables que je vais écrire
IF MesDataExd.MesData.OUT_CmdP THEN
MesDataExd.MesData.OUT_SetptP		:= MIN(MAX(IN_SetptP, MesDataExd.MesData.OUT_SetptPMin), MesDataExd.MesData.OUT_SetptPMax);
ELSE
MesDataExd.MesData.OUT_SetptP 		:= 0;
END_IF

IF MesDataExd.MesData.OUT_CmdQ THEN
MesDataExd.MesData.OUT_SetptQ		:= -MIN(MAX(IN_SetptQ, MesDataExd.MesData.OUT_SetptQMin), MesDataExd.MesData.OUT_SetptQMax);
ELSE
MesDataExd.MesData.OUT_SetptQ 		:= 0;
END_IF

MesData.OUT_SetptV := IN_SetptU;
MesData.OUT_SetptF := IN_SetptF;


TON_CmdQ_On				(IN := MesDataExd.MesData.OUT_CmdQ 					AND NOT MesDataExd.MesData.MesOpeFlag.4, PT := ParamTimeoutCmdQ);		
TON_CmdCosPhi_On		(IN := MesDataExd.MesData.OUT_CmdCosPhi 				AND NOT MesDataExd.MesData.MesOpeFlag.5, PT := ParamTimeoutCmdCosPhi);		
TON_CmdQ_Off			(IN :=  NOT MesDataExd.MesData.OUT_CmdQ  				AND MesDataExd.MesData.MesOpeFlag.4, PT := ParamTimeoutCmdQ);				   	
TON_CmdCosPhi_Off		(IN :=  NOT MesDataExd.MesData.OUT_CmdCosPhi 			AND MesDataExd.MesData.MesOpeFlag.5, PT := ParamTimeoutCmdCosPhi);		
TON_CmdBlackStart		(IN := MesDataExd.MesData.OUT_CmdBlackStart 			AND NOT MesDataExd.MesData.MesOpeFlag.8, PT := ParamTimeOutBlckStrt);
TON_FreqReg_On			(IN := MesDataExd.MesData.OUT_CmdFreqregMode 			AND NOT MesDataExd.MesData.MesOpeFlag.2, PT := ParamTimeoutPvF);			
TON_FreqReg_Off			(IN :=  NOT MesDataExd.MesData.OUT_CmdFreqregMode 		AND MesDataExd.MesData.MesOpeFlag.2, PT := ParamTimeoutPvF	);		
TON_UReg_On				(IN := MesDataExd.MesData.OUT_CmdUregMode 			AND NOT MesDataExd.MesData.MesOpeFlag.1, PT := ParamTimeoutQvU	);		
TON_UReg_Off			(IN :=  NOT MesDataExd.MesData.OUT_CmdUregMode 		AND MesDataExd.MesData.MesOpeFlag.1, PT := ParamTimeoutQvU	);		
TON_CmdGridFormer		(IN := MesDataExd.MesData.OUT_CmdGridMode 			AND NOT MesDataExd.MesData.MesOpeFlag.10, PT := ParamTimeoutGridFormerTransition	);		
TON_CmdGridFeeder		(IN :=  NOT MesDataExd.MesData.OUT_CmdGridMode			AND MesDataExd.MesData.MesOpeFlag.10, PT := ParamTimeoutGridFeederTransition	);		
TON_CmdStop				(IN := MesDataExd.MesData.OUT_CmdStop					AND MesDataExd.MesData.MesState.0);
END_METHOD

METHOD M_Init

VAR 

END_VAR
SUPER^.M_Init() ; 

MesData.OUT_CmdP := TRUE;
MesData.OUT_CmdQ := TRUE;

MesCP_Read := TRUE;
MesCP_Write := TRUE;
END_METHOD

METHOD M_Read
//////////////////
//  Read Modbus Variable for PCS . 
/////////////////

VAR 
	// Method local variables (reinitialized at each cycle) 
	MW 						: FB_MergeWordsToDint; 

	
	MesPsetPt_Temp 			: REAL ;
	MesQsetPt_Temp			: REAL ;
	MesPavailablePcs_Temp	: REAL;
	MesPavailable_Temp		: REAL;
	
	ComErrorPcs_Temp		: WORD;
	
	KK						: BYTE;  					// FOR Loop 
	LL						: BYTE;						// Alarm Loop

	MesPsetPtPcs_temp		: ARRAY[1..CstNbPcs_ESS_G] OF  REAL; // Setpt lu sur le module
	MesQsetPtPcs_temp		: ARRAY[1..CstNbPcs_ESS_G] OF  REAL;

	AX_Qty					: ARRAY[1..3] OF WORD := [75, 68, 68];
END_VAR
// CP-Read / Write 

MesDataExd.MesData.MesCP_Read := MesCP_Read ; 
MesDataExd.MesData.MesCP_Write := MesCP_Write ;  

IF MesCP_Read  THEN	
// MODBUS REQUEST//

		ModbusRead[4]
		(
			tTimeout		:= ParamTimeout,
			nUnitID			:= ParamUnitID,
			sIPAddr			:= ParamIPAddress ,
			ClockRead		:= ClockRead AND MesCP_Read,
			nTcpPort		:= ParamTcpPort,
			nQuantity		:= 75,
			Reset			:= IN_CmdReset,
			nMBAddr			:= 1100  ,//Access every PCS power modules
			cbLength		:= SIZEOF(MesBlock1_Temp[4]) , 
			pDestAddr		:= ADR(MesBlock1_Temp[4]),
			ModbusReadAlarm	=>MesModbusReadAlarm[4]
		);
    
		
		
		
// MODBUS REQUEST//
	FOR KK:=1 TO ParamNbPcs DO 	
		ModbusRead[KK]
		(
			tTimeout		:= ParamTimeout,
			nUnitID			:= ParamUnitID,
			sIPAddr			:= ParamIPAddress_DSP[KK] ,
			ClockRead		:= ClockRead AND MesCP_Read,
			nTcpPort		:= ParamTcpPort,
			nQuantity		:= AX_Qty[KK],
			Reset			:= IN_CmdReset,
			nMBAddr			:= 1000 ,
			cbLength		:= SIZEOF(MesBlock1_Temp[KK]) , 
			pDestAddr		:= ADR(MesBlock1_Temp[KK]),
			ModbusReadAlarm	=>MesModbusReadAlarm[KK]
		);
    
	END_FOR

	
	
	
// MODBUS BLOCK SEPARATION/
	// Block1 (PCS) 
	FOR KK:=1 TO ParamNbPcs DO 	// Value per Power Column (3 per inverter IBX3)
		// Measurements
		MW( WORD_STRONG:= MesBlock1_Temp[KK][1], SIGNED:=TRUE, FIX:=1 , SIZE:=1, VAR_OUT := MesDataExd.AX_PowerCol[KK].MesUdc); 
		MW( WORD_STRONG:= MesBlock1_Temp[KK][2], SIGNED:=TRUE, FIX:=1 , SIZE:=1, VAR_OUT := MesDataExd.AX_PowerCol[KK].MesIdc); //Vérifier les signes
		MW( WORD_STRONG:= MesBlock1_Temp[KK][3], SIGNED:=FALSE, FIX:=1 , SIZE:=1, VAR_OUT := MesDataExd.AX_PowerCol[KK].MesU);
		MW( WORD_STRONG:= MesBlock1_Temp[KK][6], SIGNED:=FALSE, FIX:=1 , SIZE:=1, VAR_OUT := MesDataExd.AX_PowerCol[KK].MesI1); //Vérifier les signes
		MW( WORD_STRONG:= MesBlock1_Temp[KK][7], SIGNED:=FALSE, FIX:=1 , SIZE:=1, VAR_OUT := MesDataExd.AX_PowerCol[KK].MesI2); //Vérifier les signes
		MW( WORD_STRONG:= MesBlock1_Temp[KK][8], SIGNED:=FALSE, FIX:=1 , SIZE:=1, VAR_OUT := MesDataExd.AX_PowerCol[KK].MesI3); //Vérifier les signes
		MW( WORD_STRONG:= MesBlock1_Temp[KK][9], SIGNED:=TRUE, FIX:=1 , SIZE:=1, VAR_OUT := MesDataExd.AX_PowerCol[KK].MesPdc); // Vérifier les signes
		MW( WORD_STRONG:= MesBlock1_Temp[KK][10], SIGNED:=TRUE, FIX:=1 , SIZE:=1, VAR_OUT := MesDataExd.AX_PowerCol[KK].MesP); // Vérifier les signes
		MW( WORD_STRONG:= MesBlock1_Temp[KK][11], SIGNED:=TRUE, FIX:=1 , SIZE:=1, VAR_OUT := MesDataExd.AX_PowerCol[KK].MesQ);// Vérifier les signes
		MW( WORD_STRONG:= MesBlock1_Temp[KK][12], SIGNED:=FALSE, FIX:=3 , SIZE:=1, VAR_OUT := MesDataExd.AX_PowerCol[KK].MesCosPhi);
		MW( WORD_STRONG:= MesBlock1_Temp[KK][13], SIGNED:=FALSE, FIX:=2 , SIZE:=1, VAR_OUT := MesDataExd.AX_PowerCol[KK].MesFreq);
		
		// Inputs (Temp and IO)
		MW( WORD_STRONG:= MesBlock1_Temp[KK][15], SIGNED:=TRUE, FIX:=1 , SIZE:=1, VAR_OUT := MesDataExd.AX_PowerCol[KK].MesTempControl);
		MW( WORD_STRONG:= MesBlock1_Temp[KK][18], SIGNED:=TRUE, FIX:=1 , SIZE:=1, VAR_OUT := MesDataExd.AX_PowerCol[KK].MesTempPowerUnit);

		// Alarms
	MesDataExd.AX_PowerCol[KK].MesRegAlarm0:=MesBlock1_Temp[KK][24];
	MesDataExd.AX_PowerCol[KK].MesRegAlarm1:=MesBlock1_Temp[KK][25];
	MesDataExd.AX_PowerCol[KK].MesRegAlarm2:=MesBlock1_Temp[KK][26];
	MesDataExd.AX_PowerCol[KK].MesRegAlarm3:=MesBlock1_Temp[KK][27];
	MesDataExd.AX_PowerCol[KK].MesRegAlarm4:=MesBlock1_Temp[KK][28];					

		MW( WORD_STRONG:= MesBlock1_Temp[KK][48], SIGNED:=TRUE, FIX:=1 , SIZE:=1, VAR_OUT := MesDataExd.AX_PowerCol[KK].MesTempCabinet);
		
		// States
	MesDataExd.AX_PowerCol[KK].MesAcSwitchClosed := MesBlock1_Temp[KK][61].2 ;	// AC contactor status
	MesDataExd.AX_PowerCol[KK].MesDoorOpened := NOT MesBlock1_Temp[KK][61].6; // Door : 1= Close, O= Open
	MesDataExd.AX_PowerCol[KK].MesDeratingWord := MesBlock1_Temp[KK][62] ;
		
		MW( WORD_STRONG:= MesBlock1_Temp[KK][68], SIGNED:=FALSE, FIX:=0 , SIZE:=1, VAR_OUT := MesDataExd.AX_PowerCol[KK].MesHeartbit);
		

	END_FOR

	// Inverter states (à tester)

MesDataExd.MesData.MesOpeFlag					:= MesBlock1_Temp[4][67];
MesDataExd.MesData.MesSnom						:= ParamSmax;		//MàJ : WORD_TO_REAL(MesBlock1_Temp[1][69]);
MesDataExd.MesData.MesAvailability				:= WORD_TO_REAL(MesBlock1_Temp[4][70]);
	
	MW( WORD_STRONG := MesBlock1_Temp[4][71], SIZE := 1, FIX := 0, SIGNED := FALSE, VAR_OUT := MesDataExd.MesData.MesHumidity);
	MW( WORD_STRONG := MesBlock1_Temp[4][72], SIZE := 1, FIX := 1, SIGNED := TRUE, VAR_OUT := MesDataExd.MesData.MesTemp);
	
MesDataExd.MesData.MesPrecharge 				:= WORD_TO_BOOL(MesBlock1_Temp[4][73]);
MesDataExd.MesData.MesDcBreaker				:= MesBlock1_Temp[4][74].0;
MesDataExd.MesData.MesAcBreaker				:= MesBlock1_Temp[4][61].0;
MesDataExd.MesData.MesSoCLimitReached			:= MesBlock1_Temp[4][74].2;
MesDataExd.MesData.MesOffGrid					:= MesBlock1_Temp[4][74].3;
MesDataExd.MesData.MesOnGrid					:= MesBlock1_Temp[4][74].4;
MesDataExd.MesData.MesHeartBeat				:= MesBlock1_Temp[4][75];
END_IF
END_METHOD

METHOD M_StateManager
//////////////////
// Detect which is the state of the PCS system . 
/////////////////

VAR 
	// Method local variables (reinitialized at each cycle) 

	
END_VAR
 MesDataExd.MesData.MesState 		:= 0;



IF NOT MesDataExd.MesData.MesAcBreaker AND NOT MesDataExd.MesData.MesDcBreaker THEN 
	// OFF State :  No Charger connected or all charger in alarm
MesDataExd.MesData.MesState.0 	:= 1 ; 
	
ELSIF MesDataExd.MesData.MesOffGrid THEN
	// Feeding master
MesDataExd.MesData.MesState.1 	:= 1 ; 
	
ELSIF MesDataExd.MesData.MesOnGrid THEN
	// Feeding slave
MesDataExd.MesData.MesState.2 	:= 1 ; 
	
END_IF

SUPER^.M_StateManager() ;
END_METHOD

METHOD M_WriteCommand
//////////////////
//  Modbus Write of the command for the PCS. 
/////////////////

VAR 
	// Method local variables (reinitialized at each cycle) 
	
	AX_Adr			: ARRAY[1..3] OF UINT := [1707	, 1802	, 	0217	];
	AX_QTY			: ARRAY[1..3] OF BYTE := [40	, 33	, 	2		];
	AX_UnitID		: ARRAY[1..3] OF BYTE := [1		, 1		, 	1		];	

	KK: INT;
	
END_VAR

TRIG_CmdP_On			(CLK := IN_CmdP_On);						
TRIG_CmdP_Off			(CLK := IN_CmdP_Off);							
TRIG_CmdQ_On			(CLK := IN_CmdQ_On);                        
TRIG_CmdQ_Off			(CLK := IN_CmdQ_Off);                      
TRIG_CmdCosPhi_On		(CLK := IN_CmdCosPhi_On);              
TRIG_CmdCosPhi_Off		(CLK := IN_CmdCosPhi_Off);            
TRIG_CmdReset			(CLK := IN_CmdReset);
TRIG_FreqReg_On			(CLK := IN_CmdFreqregOn);
TRIG_FreqReg_Off		(CLK := IN_CmdFreqregOff);
TRIG_UReg_On			(CLK := IN_CmdUregOn);			
TRIG_UReg_Off			(CLK := IN_CmdUregOff);
TRIG_CmdGridFormer		(CLK := IN_CmdGridFormer);
TRIG_CmdGridFeeder		(CLK := IN_CmdGridFeeder);
TRIG_CmdMicroCyclingOn	(CLK := IN_CmdMicroCyclingOn AND MesMicroCyclingAllowed);
TRIG_CmdMicroCyclingOff	(CLK := IN_CmdMicroCyclingOff OR Trig_MicroCyclingNoLongerAllowed.Q);	
TRIG_CmdOpenAC			(CLK := IN_CmdOpenAC);
TRIG_CmdOpenDC			(CLk := IN_CmdOpenDC);
TRIG_CmdStop			(CLK := IN_CmdStop);
TRIG_CmdStandby			(CLK := IN_CmdStandby  AND NOT TP_CmdStop.Q );
TRIG_CmdStart			(CLK := IN_CmdStart AND NOT TP_CmdStop.Q AND NOT IN_CmdStopOperation AND NOT IN_CmdPreventStart);
TRIG_CmdBlackStart		(CLK := IN_CmdBlackStart);	
TRIG_CmdPcsLocal		(CLk := IN_CmdInvLocal);
TRIG_LowLowSoC			(clk := DataSystemBMS.MesSoCConnected <= A1_PP.ParamSocVeryVeryLow);
	
TP_CmdPreStop	(IN := TRIG_CmdStop.Q, 												PT := T#1S500MS);
TP_CmdPreStart	(IN := TRIG_CmdStart.Q, 											PT := ParamTimePulseTrig);
TP_CmdOpenAC	(IN := TRIG_CmdOpenAC.Q, 											PT := ParamTimePulseTrig);
TP_CmdOpenDC	(IN := TRIG_CmdOpenDC.Q, 											PT := ParamTimePulseTrig);
TP_CmdStop		(IN := F_TrigPreStop.Q, 											PT := ParamTimePulseTrig);
TP_CmdStart		(IN := F_TrigPreStart.Q, 											PT := ParamTimePulseTrig);
TP_CmdStandby	(IN := TRIG_CmdStop.Q OR TRIG_CmdStandby.Q OR TRIG_LowLowSoC.Q, 	PT := ParamTimePulseTrig);
TP_Reset		(IN := TRIG_CmdReset.Q, 											PT := ParamTimePulseTrig);


F_TrigPreStart	(CLK := TP_CmdPreStart.Q);
F_TrigPreStop	(CLK := TP_CmdPreStop.Q);


IF TRIG_CmdBlackStart.Q THEN
	IN_CmdBlackStart := FALSE;
END_IF
IF TRIG_CmdStop.Q THEN
	IN_CmdStop := FALSE;
END_IF
IF TRIG_CmdStart.Q THEN
	AX_ESS[ParamEssNum].AX_BAT[ParamPcsNum].IN_CmdCloseDC := TRUE;
	IN_CmdStart := FALSE;
END_IF
IF TRIG_CmdStandby.Q THEN
	IN_CmdStandby := FALSE;
END_IF

IF TRIG_CmdReset.Q THEN
	IN_CmdReset := FALSE;
END_IF

IF TRIG_CmdP_Off.Q THEN
MesDataExd.MesData.OUT_CmdP := FALSE;
	IN_CmdP_Off := FALSE;
END_IF
IF TRIG_CmdP_On.Q THEN
MesDataExd.MesData.OUT_CmdP := TRUE;
	IN_CmdP_On := FALSE;
END_IF
IF TRIG_CmdQ_Off.Q OR TRIG_CmdCosPhi_On.Q THEN
MesDataExd.MesData.OUT_CmdQ := FALSE;
	IN_CmdQ_Off := FALSE;
END_IF
IF TRIG_CmdQ_On.Q THEN
MesDataExd.MesData.OUT_CmdQ := TRUE;
	IN_CmdQ_On := FALSE;
END_IF
IF TRIG_CmdCosPhi_Off.Q OR TRIG_CmdQ_On.Q THEN
MesDataExd.MesData.OUT_CmdCosPhi := FALSE;
	IN_CmdCosPhi_Off := FALSE;
END_IF
IF TRIG_CmdCosPhi_On.Q THEN
MesDataExd.MesData.OUT_CmdCosPhi := TRUE;
MesDataExd.MesData.OUT_SetptCosPhi	:= IN_SetptCosPhi;
	IN_CmdCosPhi_On := FALSE;
END_IF

IF TRIG_FreqReg_On.Q THEN
MesDataExd.MesData.OUT_CmdFreqregMode := TRUE;
	IN_CmdFreqregOn := FALSE;
END_IF
IF TRIG_FreqReg_Off.Q THEN
MesDataExd.MesData.OUT_CmdFreqregMode := FALSE;
	IN_CmdFreqregOff := FALSE;
END_IF

IF TRIG_UReg_On.Q THEN
MesDataExd.MesData.OUT_CmdUregMode := TRUE;
	IN_CmdUregOn := FALSE;
END_IF
IF TRIG_UReg_Off.Q THEN
MesDataExd.MesData.OUT_CmdUregMode := FALSE;
	IN_CmdUregOff := FALSE;
END_IF
	
IF TRIG_CmdGridFormer.Q THEN
MesDataExd.MesData.OUT_CmdGridMode := TRUE;
	IN_CmdGridFormer := FALSE;
END_IF 
IF TRIG_CmdGridFeeder.Q OR TRIG_CmdStop.Q THEN //Si on fait une commande stop, on passe le mode en grid feeder
MesDataExd.MesData.OUT_CmdGridMode := FALSE;
	IN_CmdGridFeeder := FALSE;
END_IF

IF TRIG_CmdMicroCyclingOn.Q THEN
	IF DataSystemBMS.MesSoC > ParamMicroCyclingSoCMax *0.95 THEN
		MesMicroCyclingP := ABS(ParamMicroCyclingPower);
	ELSE
		MesMicroCyclingP := -ABS(ParamMicroCyclingPower);
	END_IF
	
	IN_CmdMicroCyclingOn := FALSE;
MesDataExd.MesData.OUT_CmdMicroCyclingMode := TRUE;
END_IF 
IF TRIG_CmdMicroCyclingOff.Q THEN
	IN_CmdMicroCyclingOff := FALSE;
MesDataExd.MesData.OUT_CmdMicroCyclingMode := FALSE;
END_IF 

IF TRIG_CmdPcsLocal.Q THEN
	IN_CmdInvLocal := FALSE;
MesDataExd.MesData.OUT_CmdInvLocal := NOT MesDataExd.MesData.OUT_CmdInvLocal;
END_IF

IN_CmdWatchdog := CalLocalTimeStruct.wSecond MOD 2 = 0;

MesData.OUT_CmdStop 		:= TP_CmdStop.Q;
MesData.OUT_CmdStart 		:= TP_CmdStart.Q;
MesData.OUT_CmdBlackStart 	:= TP_CmdBlackStart.Q;
MesData.OUT_CmdStandby 		:= TP_CmdStandby.Q;


Trig_Write[1](CLK := MEMCMP(pBuf1 :=ADR(AX_Cmd[1]), pBuf2 := ADR(AX_Cmd_Old[1]), n := SIZEOF(AX_CMD[1]))<>0);
Trig_Write[2](CLK := MEMCMP(pBuf1 :=ADR(AX_Cmd[2]), pBuf2 := ADR(AX_Cmd_Old[2]), n := SIZEOF(AX_CMD[2]))<>0);
Trig_Write[3](CLK := MEMCMP(pBuf1 :=ADR(AX_Cmd[3]), pBuf2 := ADR(AX_Cmd_Old[3]), n := SIZEOF(AX_CMD[3]))<>0);

IF MEMCMP(pBuf1 :=ADR(AX_Cmd[1]), pBuf2 := ADR(AX_Cmd_Old[1]), n := SIZEOF(AX_CMD[1]))<>0 THEN
	MEMCPY(destAddr := ADR(AX_Cmd_Old[1]), srcAddr := ADR(AX_Cmd[1]), n:= SIZEOF(AX_Cmd[1]));
END_IF
IF MEMCMP(pBuf1 :=ADR(AX_Cmd[2]), pBuf2 := ADR(AX_Cmd_Old[2]), n := SIZEOF(AX_CMD[2]))<>0 THEN
	MEMCPY(destAddr := ADR(AX_Cmd_Old[2]), srcAddr := ADR(AX_Cmd[2]), n:= SIZEOF(AX_Cmd[2]));
END_IF		
IF MEMCMP(pBuf1 :=ADR(AX_Cmd[3]), pBuf2 := ADR(AX_Cmd_Old[3]), n := SIZEOF(AX_CMD[3]))<>0 THEN
	MEMCPY(destAddr := ADR(AX_Cmd_Old[3]), srcAddr := ADR(AX_Cmd[3]), n:= SIZEOF(AX_Cmd[3]));
END_IF			

	// Manouvers (41708)
		AX_Cmd[1][1].1:= IN_CmdOpenAC;
		AX_Cmd[1][1].2:= IN_CmdOpenDC;
		
	// SoC	
		AX_Cmd[1][2]  := REAL_TO_WORD(ParamFreqRegSoCmax); 
		AX_Cmd[1][3]  := REAL_TO_WORD(ParamFreqRegSoCmin); 
		AX_Cmd[1][4]  := REAL_TO_WORD(TRUNC(DataSystemBMS.MesSoCConnected));		// SoC connected 
		
		
